(******************************************************************************************************************************************)
(****************************				           Reset Function Part                                                 *****************************)
(******************************************************************************************************************************************)
IF xReset AND NOT(xSetEnd) THEN
	xEnd:=FALSE;
	xSetEnd:=TRUE;
END_IF;
(******************************************************************************************************************************************)
(****************************				              Error Controlling Part                                            *****************************)
(******************************************************************************************************************************************)
IF (xHardwareError OR ((TAxisGrindFeeder.T_CtrleSingle.xErr) AND xStartMainPrc)) AND NOT(xSetEnd) THEN
	IF NOT(TAxisGrindFeeder.T_CtrleSingle.xExecute) THEN
		IF NOT(xInitError) THEN
			iStepError:=100;
			xInitError:=TRUE;
			IF xHardwareError THEN
				iErrorNr:=iTmpErrorNr;
			ELSE
				xHardwareError:=TRUE;	(* Hardware Error *)
			END_IF;
		END_IF;
		CASE iStepError OF
			100:	iStepError:=0;
				xError:=TRUE;
		END_CASE;
		IF xQuitErr THEN
			xSetEnd:=TRUE;
		END_IF;
	END_IF;
END_IF;
(******************************************************************************************************************************************)
(****************************				              Main Controlling Part                                            *****************************)
(******************************************************************************************************************************************)
IF (xStart OR xStartMainCtr) AND NOT(xSetEnd) AND NOT(xHardwareError) THEN
	IF NOT (xInitMainCtr) THEN
		iTmpErrorNr:=0;
		iStepPrc:=100;
		xInitMainCtr:=TRUE;
		xStartMainCtr:=TRUE;
		xStart:=FALSE;
		xEnd:=FALSE;
		xAbord:=FALSE;
		xTmpInit:=FALSE;
	END_IF;
	IF xStop AND NOT(xTmpInit) THEN
		xTmpInit:=TRUE;
		iTmp:=100;
		RETURN;
	END_IF;
	IF xFreeze THEN
		IF xStart AND NOT(xAbord) THEN
			xFreeze:=FALSE;
			xStart:=FALSE;
		END_IF;
		IF xAbord THEN
			xAbord:=FALSE;
			xFreeze:=FALSE;
			xStart:=FALSE;
			xSetEnd:=TRUE;
		END_IF;
		RETURN;
	END_IF;
	IF NOT(xStartMainPrc) AND NOT(xSetEnd) THEN
		xStartMainPrc:=TRUE;
	END_IF;
END_IF;
(******************************************************************************************************************************************)
(****************************				             immediate Stop Part                                              *****************************)
(******************************************************************************************************************************************)
IF xTmpInit AND NOT(xSetEnd) THEN
	IF NOT(xSafetyCircuitOn) THEN
		xTmpInit:=FALSE;
		iTmp:=100;
		xSetEnd:=TRUE;
		RETURN;
	END_IF;
	CASE iTmp OF
		100:	TAxisGrindFeeder.T_CtrleSingle.iFunction:=5;
			TAxisGrindFeeder.T_CtrleSingle.xExecute:=TRUE;
			iTmp:=200;
			RETURN;
		200:	IF NOT(TAxisGrindFeeder.T_CtrleSingle.xExecute) AND TAxisGrindFeeder.T_CtrleSingle.xDone THEN
				iTmp:=300;
			END_IF;
			RETURN;
		300:	xTmpInit:=FALSE;
			iTmp:=100;
			xSetEnd:=TRUE;
			RETURN;
	END_CASE;
END_IF;
(******************************************************************************************************************************************)
(****************************				             Main Procedure Part                                             *****************************)
(******************************************************************************************************************************************)
IF xStartMainPrc AND NOT(xSetEnd) AND NOT(xHardwareError) THEN
	CASE iStepPrc OF
		100:	IF NOT(xInitStep) THEN
				xInitStep:=TRUE;
				IF NOT(TAxisGrindFeeder.T_CtrleSingle.xDone)THEN
					xHardwareError:=TRUE;
					iTmpErrorNr:=1;
					RETURN;
				END_IF;
				IF NOT(TAxisGrindFeeder.T_CtrleSingle.xPower) THEN
					TAxisGrindFeeder.T_CtrleSingle.iFunction:=3;
					TAxisGrindFeeder.T_CtrleSingle.xExecute:=TRUE;
				END_IF;
			END_IF;
			IF NOT(TAxisGrindFeeder.T_CtrleSingle.xExecute) AND TAxisGrindFeeder.T_CtrleSingle.xDone THEN
				xStartMainPrc:=FALSE;
				xInitStep:=FALSE;
				iStepPrc:=200;
			END_IF;
		200:	IF NOT(xInitStep) THEN
				xInitStep:=TRUE;
				IF (iFunctionNr = 4) THEN
					TAxisGrindFeeder.T_CtrleSingle.iFunction:=7;	(* Move Absolut *)
				END_IF;
				IF (iFunctionNr = 5) THEN
					TAxisGrindFeeder.T_CtrleSingle.iFunction:=8;	(* Move Relative *)
				END_IF;
				TAxisGrindFeeder.T_CtrleSingle.xExecute:=TRUE;
			END_IF;
			IF NOT(TAxisGrindFeeder.T_CtrleSingle.xExecute) AND TAxisGrindFeeder.T_CtrleSingle.xDone THEN
				xStartMainPrc:=FALSE;
				xInitStep:=FALSE;
				iStepPrc:=0;
				xSetEnd:=TRUE;
			END_IF;
	END_CASE;
END_IF;
(******************************************************************************************************************************************)
(****************************				           Parallel Procedure Part                                          *****************************)
(******************************************************************************************************************************************)

(******************************************************************************************************************************************)
(****************************				             	Init / Reset Part                                                   *****************************)
(******************************************************************************************************************************************)
IF xSetEnd THEN
	xEnd:=TRUE;
	xInitStep:=FALSE;
	xSetEnd:=FALSE;
	xStop:=FALSE;
	xStartMainPrc:=FALSE;
	xInitMainCtr:=FALSE;
	xStartMainCtr:=FALSE;
	xStart:=FALSE;
	xHardwareError:=FALSE;
	xQuitErr:=FALSE;
	xError:=FALSE;
	iErrorNr:=0;
	xInitError:=FALSE;
	xFreeze:=FALSE;
	xAbord:=FALSE;
	xReset:=FALSE;
END_IF;
END_FUNCTION_BLOCK

(* POU PRG_STATION_LAYER3/FB_STATIONEN/FB_FUNCTION/FB_FctSetAxisPosition, ST *)
FUNCTION_BLOCK FB_FctSetAxisPosition
VAR_INPUT
	xMicroRodActive: BOOL;		(* choice of the machine MicroWire or MicroRod *)
	xBeckhoffDriveActive: BOOL;	(* choice of the axis Beckhoff or EcoStep *)
	xSafetyCircuitOn:BOOL;			(* state of the safety circuit-->TRUE=Machine current ON, FALSE=Machine current OFF *)
	iFunctionNr:INT;				(* state of the called function number-->	6=set position of the ToolLeft axis
																	7=set position of the ToolCenter axis
																	8=set position of the ToolRight axis
																	9=set position of the ToolFeeder axis
																	10=set position of the GrindFeeder axis *)
END_VAR
VAR_IN_OUT
	xStart : BOOL;					(* start the function *)
	xReset : BOOL;				(* reset the function *)
	xStop : BOOL;					(* stop the active function *)
	xQuitErr : BOOL;				(* quit the error caused of the active function *)
	xAbord : BOOL;				(* abord the active function *)
	TAxisToolLeft:ST_AXIS;		(* data structure for the ToolLeft axis *)
	TAxisToolCenter:ST_AXIS;		(* data structure for the ToolCenter axis *)
	TAxisToolRight:ST_AXIS;		(* data structure for the ToolRight axis *)
	TAxisToolFeeder:ST_AXIS;		(* data structure for the ToolFeeder axis *)
	TAxisGrindFeeder:ST_AXIS;	(* data structure for the GrindFeeder axis *)
END_VAR
VAR_OUTPUT
	xEnd : BOOL;					(* state of the function if a active function is ended *)
	xError : BOOL;					(* state of the function if a active function caused an error *)
	iErrorNr : INT;					(* state of the function if a active function caused an error, in this case give the error number *)
END_VAR
VAR
	xHardwareError: BOOL := FALSE;
	xInitError: BOOL := FALSE;
	iStepError: INT := 0;
	xStartMainCtr: BOOL := FALSE;
	xStartMainPrc: BOOL := FALSE;
	xInitMainCtr: BOOL := FALSE;
	iStepPrc: INT := 0;
	xSetEnd: BOOL := FALSE;
	xInitStep: BOOL := FALSE;
	xFreeze: BOOL := FALSE;
	iTmpErrorNr:INT:=0;
	xTmpInit:BOOL;
	iTmp:INT;
	ptrTAxis: POINTER TO ST_AXIS;
	xReadFirstTime: BOOL;
END_VAR
(****************************************************************************************************************************************************)
(***********       This Functionblock set a position for the ToolLeft,ToolCenter,ToolRight,ToolFeeder or GrindFeeder       ************)
(****************************************************************************************************************************************************)

IF NOT(xReadFirstTime) THEN
	xReadFirstTime:=TRUE;
	ptrTAxis:=ADR(TAxisToolLeft);
END_IF;
(******************************************************************************************************************************************)
(****************************				           Reset Function Part                                                 *****************************)
(******************************************************************************************************************************************)
IF xReset AND NOT(xSetEnd) THEN
	ptrTAxis:=ADR(TAxisToolLeft);
	xEnd:=FALSE;
	xSetEnd:=TRUE;
END_IF;
(******************************************************************************************************************************************)
(****************************				              Error Controlling Part                                            *****************************)
(******************************************************************************************************************************************)
IF (xHardwareError OR ((ptrTAxis^.T_CtrleSingle.xErr) AND xStartMainPrc)) AND NOT(xSetEnd) THEN
	IF NOT(ptrTAxis^.T_CtrleSingle.xExecute) THEN
		IF NOT(xInitError) THEN
			iStepError:=100;
			xInitError:=TRUE;
			IF xHardwareError THEN
				iErrorNr:=iTmpErrorNr;
			ELSE
				xHardwareError:=TRUE;	(* Hardware Error *)
			END_IF;
		END_IF;
		CASE iStepError OF
			100:	iStepError:=0;
				xError:=TRUE;
		END_CASE;
		IF xQuitErr THEN
			xSetEnd:=TRUE;
		END_IF;
	END_IF;
END_IF;
(******************************************************************************************************************************************)
(****************************				              Main Controlling Part                                            *****************************)
(******************************************************************************************************************************************)
IF (xStart OR xStartMainCtr) AND NOT(xSetEnd) AND NOT(xHardwareError) THEN
	IF NOT (xInitMainCtr) THEN
		IF (iFunctionNr = 6) THEN
			ptrTAxis:=ADR(TAxisToolLeft);
		ELSIF (iFunctionNr = 7) THEN
			ptrTAxis:=ADR(TAxisToolCenter);
		ELSIF (iFunctionNr = 8) THEN
			ptrTAxis:=ADR(TAxisToolRight);
		ELSIF (iFunctionNr = 9) THEN
			ptrTAxis:=ADR(TAxisToolFeeder);
		ELSIF (iFunctionNr = 10) THEN
			ptrTAxis:=ADR(TAxisGrindFeeder);
		ELSE
			ptrTAxis:=ADR(TAxisToolLeft);
		END_IF;
		iTmpErrorNr:=0;
		iStepPrc:=100;
		xInitMainCtr:=TRUE;
		xStartMainCtr:=TRUE;
		xStart:=FALSE;
		xEnd:=FALSE;
		xAbord:=FALSE;
		xTmpInit:=FALSE;
	END_IF;
	IF xStop AND NOT(xTmpInit) THEN
		xTmpInit:=TRUE;
		iTmp:=100;
		RETURN;
	END_IF;
	IF xFreeze THEN
		IF xStart AND NOT(xAbord) THEN
			xFreeze:=FALSE;
			xStart:=FALSE;
		END_IF;
		IF xAbord THEN
			xAbord:=FALSE;
			xFreeze:=FALSE;
			xStart:=FALSE;
			xSetEnd:=TRUE;
		END_IF;
		RETURN;
	END_IF;
	IF NOT(xStartMainPrc) AND NOT(xSetEnd) THEN
		xStartMainPrc:=TRUE;
	END_IF;
END_IF;
(******************************************************************************************************************************************)
(****************************				             immediate Stop Part                                              *****************************)
(******************************************************************************************************************************************)
IF xTmpInit AND NOT(xSetEnd) THEN
	IF NOT(xSafetyCircuitOn) THEN
		xTmpInit:=FALSE;
		iTmp:=100;
		xSetEnd:=TRUE;
		RETURN;
	END_IF;
	CASE iTmp OF
		100:	IF NOT(ptrTAxis^.T_CtrleSingle.xDone) THEN
				ptrTAxis^.T_CtrleSingle.xReset:=TRUE;
				iTmp:=200;
			END_IF;
			RETURN;
		200:	IF NOT(ptrTAxis^.T_CtrleSingle.xReset) AND ptrTAxis^.T_CtrleSingle.xDone THEN
				iTmp:=300;
			END_IF;
			RETURN;
		300:	xTmpInit:=FALSE;
			iTmp:=100;
			xSetEnd:=TRUE;
			RETURN;
	END_CASE;
END_IF;
(******************************************************************************************************************************************)
(****************************				             Main Procedure Part                                             *****************************)
(******************************************************************************************************************************************)
IF xStartMainPrc AND NOT(xSetEnd) AND NOT(xHardwareError) THEN
	CASE iStepPrc OF
		100:	IF NOT(xInitStep) THEN
				xInitStep:=TRUE;
				IF NOT(ptrTAxis^.T_CtrleSingle.xDone)THEN
					xHardwareError:=TRUE;
					iTmpErrorNr:=1;
					RETURN;
				END_IF;
				ptrTAxis^.T_CtrleSingle.iFunction:=11;
				ptrTAxis^.T_CtrleSingle.xExecute:=TRUE;
			END_IF;
			IF NOT(ptrTAxis^.T_CtrleSingle.xExecute) AND ptrTAxis^.T_CtrleSingle.xDone THEN
				xStartMainPrc:=FALSE;
				xInitStep:=FALSE;
				iStepPrc:=0;
				xSetEnd:=TRUE;
			END_IF;
	END_CASE;
END_IF;
(******************************************************************************************************************************************)
(****************************				           Parallel Procedure Part                                          *****************************)
(******************************************************************************************************************************************)

(******************************************************************************************************************************************)
(****************************				             	Init / Reset Part                                                   *****************************)
(******************************************************************************************************************************************)
IF xSetEnd THEN
	xEnd:=TRUE;
	xInitStep:=FALSE;
	xSetEnd:=FALSE;
	xStop:=FALSE;
	xStartMainPrc:=FALSE;
	xInitMainCtr:=FALSE;
	xStartMainCtr:=FALSE;
	xStart:=FALSE;
	xHardwareError:=FALSE;
	xQuitErr:=FALSE;
	xError:=FALSE;
	iErrorNr:=0;
	xInitError:=FALSE;
	xFreeze:=FALSE;
	xAbord:=FALSE;
	xReset:=FALSE;
END_IF;
END_FUNCTION_BLOCK

(* POU PRG_STATION_LAYER3/FB_STATIONEN/FB_FUNCTION/FB_FctToolWorkingGeometry, ST *)
FUNCTION_BLOCK FB_FctToolWorkingGeometry
VAR_INPUT
	xMicroRodActive: BOOL;		(* choice of the machine MicroWire or MicroRod *)
	xBeckhoffDriveActive: BOOL;	(* choice of the axis Beckhoff or EcoStep *)
	xSafetyCircuitOn:BOOL;			(* state of the safety circuit-->TRUE=Machine current ON, FALSE=Machine current OFF *)
	T_ProcessImageData:ST_RETAIN_DATA_PROCESSIMAGE;	(* Novram data structure for the process parameter *)
	T_Standard:ST_RETAIN_DATA;							(* Novram data structure for the standard process parameter *)
END_VAR
VAR_IN_OUT
	xStart : BOOL;					(* start the function *)
	xReset : BOOL;				(* reset the function *)
	xStop : BOOL;					(* stop the active function *)
	xQuitErr : BOOL;				(* quit the error caused of the active function *)
	xAbord : BOOL;				(* abord the active function *)
	TAxisToolLeft:ST_AXIS;		(* data structure for the ToolLeft axis *)
	TAxisToolCenter:ST_AXIS;		(* data structure for the ToolCenter axis *)
	TAxisToolRight:ST_AXIS;		(* data structure for the ToolRight axis *)
	TAxisToolFeeder:ST_AXIS;		(* data structure for the ToolFeeder axis *)
	TAxisGrindFeeder:ST_AXIS;	(* data structure for the GrindFeeder axis *)
	T_WorkTool:ST_WORKTOOL;	(* Tool parameter *)
END_VAR
VAR_OUTPUT
	xEnd : BOOL;					(* state of the function if a active function is ended *)
	xError : BOOL;					(* state of the function if a active function caused an error *)
	iErrorNr : INT;					(* state of the function if a active function caused an error, in this case give the error number *)
	bActivePartNumber:BYTE;		(* gives the active number of the worked section of the geometry *)
	lrProcessToolFeederActualPosition:LREAL;	(* gives the calculated position of the ToolFeeder *)
	lrProcessToolFeederSpeed:LREAL;			(* gives the calculated speed of the ToolFeeder *)
	iCountDownPlungeCycle:INT;
END_VAR
VAR
	xHardwareError: BOOL := FALSE;
	xInitError: BOOL := FALSE;
	iStepError: INT := 0;
	xStartMainCtr: BOOL := FALSE;
	xStartMainPrc: BOOL := FALSE;
	xInitMainCtr: BOOL := FALSE;
	iStepPrc: INT := 0;
	xSetEnd: BOOL := FALSE;
	xInitStep: BOOL := FALSE;
	xFreeze: BOOL := FALSE;
	iTmpErrorNr:INT:=0;
	xTmpInit:BOOL;
	iTmp:INT;
	xTmp: BOOL;
	xReadFirstTime: BOOL;
	xTmp1: BOOL;
	rToolRotationSpeed: REAL;
	FBToolCalcul:FB_TOOL_CALCUL_NEW;

	rToolFeedLength: REAL;
	rToolDiameter: REAL;
	rGrindFeedPlunge: REAL;
	ii: INT;
	iStartSection: INT;
	iEndSection: INT;
	rSpeedGrindFeed: REAL;
	rSpeedToolFeed: REAL;
	rTimeGrindPlunge: REAL;
	FBCalcGearFactor: FB_CALC_GEARFACTOR;
	lrToolFeederActualPosition: LREAL;
	iTmpStartSection: INT;
	FBCalcPlungeGrinding: FB_CALC_PLUNGE_GRINDING;
	xResetFB: BOOL;
	xGrindFeedMaster: BOOL;
	xCheckToolFeedPosition: BOOL;
	lrToolFeederPosition: LREAL;
	lrToolRightPosition: LREAL;
	lrSaveToolFeederPosition: LREAL;
	lrSaveToolRightPosition: LREAL;
	rPlungeCycleGrindFeedGeometry: REAL;
	lrGearFactor: LREAL;
	xPositionReached: BOOL;
	lrToolFeedCalcLengthPosition: REAL;
	lrCalcToolLengthInc: LREAL;
	lrCalcToolLength: LREAL;
	xReadyToolFeedStop: BOOL;
	xReadyGrindFeedStop: BOOL;
END_VAR
(****************************************************************************************************************************************************)
(***********                                This Functionblock define the function for work a geometry on the tool                                          ************)
(****************************************************************************************************************************************************)

IF NOT(xReadFirstTime) THEN
	xReadFirstTime:=TRUE;
END_IF;
(******************************************************************************************************************************************)
(****************************				           Reset Function Part                                                 *****************************)
(******************************************************************************************************************************************)
IF xReset AND NOT(xSetEnd) THEN
	xEnd:=FALSE;
	xSetEnd:=TRUE;
END_IF;
(******************************************************************************************************************************************)
(****************************				              Error Controlling Part                                            *****************************)
(******************************************************************************************************************************************)
xTmp:=	TAxisToolLeft.T_CtrleSingle.xErr OR
		(TAxisToolCenter.T_CtrleSingle.xErr AND xMicroRodActive) OR
		TAxisToolRight.T_CtrleSingle.xErr OR
		TAxisToolFeeder.T_CtrleSingle.xErr OR
		TAxisGrindFeeder.T_CtrleSingle.xErr;
xTmp1:=	NOT(TAxisToolLeft.T_CtrleSingle.xExecute) AND
		((NOT(TAxisToolCenter.T_CtrleSingle.xExecute) AND xMicroRodActive) OR NOT(xMicroRodActive)) AND
		 NOT(TAxisToolRight.T_CtrleSingle.xExecute) AND
		((NOT(TAxisToolFeeder.T_CtrleSingle.xExecute) AND NOT(xMicroRodActive)) OR xMicroRodActive) AND
		NOT(TAxisGrindFeeder.T_CtrleSingle.xExecute);
IF (xHardwareError OR (xTmp AND xStartMainPrc)) AND NOT(xSetEnd) THEN
	IF xTmp1 THEN
		IF NOT(xInitError) THEN
			iStepError:=100;
			xInitError:=TRUE;
			IF xHardwareError THEN
				iErrorNr:=iTmpErrorNr;
			ELSE
				xHardwareError:=TRUE;	(* Hardware Error *)
			END_IF;
		END_IF;
		CASE iStepError OF
			100:	iStepError:=0;
				xError:=TRUE;
		END_CASE;
		IF xQuitErr THEN
			xSetEnd:=TRUE;
		END_IF;
	END_IF;
END_IF;
(******************************************************************************************************************************************)
(****************************				              Main Controlling Part                                            *****************************)
(******************************************************************************************************************************************)
IF (xStart OR xStartMainCtr) AND NOT(xSetEnd) AND NOT(xHardwareError) THEN
	IF NOT (xInitMainCtr) THEN
		iTmpErrorNr:=0;
		iStepPrc:=100;
		xInitMainCtr:=TRUE;
		xStartMainCtr:=TRUE;
		xStart:=FALSE;
		xEnd:=FALSE;
		xAbord:=FALSE;
		xTmpInit:=FALSE;
		xCheckToolFeedPosition:=FALSE;
		bActivePartNumber:=0;
		lrCalcToolLengthInc:=lrCalcToolLength:=0.0;
		rSpeedToolFeed:=0.0;
		iCountDownPlungeCycle:=1;
	END_IF;
	IF xStop AND NOT(xTmpInit) THEN
		xTmpInit:=TRUE;
		iTmp:=100;
		RETURN;
	END_IF;
	IF xFreeze THEN
		IF xStart AND NOT(xAbord) THEN
			xFreeze:=FALSE;
			xStart:=FALSE;
		END_IF;
		IF xAbord THEN
			xAbord:=FALSE;
			xFreeze:=FALSE;
			xStart:=FALSE;
			xSetEnd:=TRUE;
		END_IF;
		RETURN;
	END_IF;
	IF NOT(xStartMainPrc) AND NOT(xSetEnd) THEN
		xStartMainPrc:=TRUE;
	END_IF;
END_IF;
(******************************************************************************************************************************************)
(****************************		               Controlling of the ToolFeeder Position                            *****************************)
(******************************************************************************************************************************************)
IF xCheckToolFeedPosition THEN
	IF xMicroRodActive THEN
		lrToolFeederPosition:=TAxisToolFeeder.T_LiveValue.lrActualPositionNotModulo - lrSaveToolFeederPosition;
		lrToolFeederActualPosition:=(lrToolFeederPosition / TAxisToolFeeder.T_CtrleSingle.lrScaleFactor);
		lrCalcToolLength:=lrToolFeederActualPosition;
	END_IF;
	IF NOT(xMicroRodActive) AND (TAxisToolRight.T_CtrleSingle.lrGearRatio <> 0.0) THEN
		lrToolFeedCalcLengthPosition:=((((T_WorkTool.rToolLength * 10.0) / ABS(T_WorkTool.rPitch)) * 24000.0) / TAxisToolRight.T_CtrleSingle.lrScaleFactor);
		lrToolFeederPosition:=lrToolFeederPosition + ABS(ABS(TAxisToolRight.T_LiveValue.lrActualPosition) - (lrSaveToolFeederPosition / TAxisToolRight.T_CtrleSingle.lrScaleFactor));
		lrSaveToolFeederPosition:=ABS(TAxisToolRight.T_LiveValue.lrActualPositionNotModulo);
		lrToolFeederActualPosition:=((T_WorkTool.rToolLength * 10.0) / lrToolFeedCalcLengthPosition) * lrToolFeederPosition;
		lrCalcToolLength:=lrCalcToolLengthInc + lrToolFeederActualPosition;
	END_IF;
ELSE
	IF NOT(xMicroRodActive) AND (TAxisToolRight.T_CtrleSingle.lrGearRatio <> 0.0) THEN
		lrSaveToolFeederPosition:=ABS(TAxisToolRight.T_LiveValue.lrActualPositionNotModulo);
		lrSaveToolRightPosition:=TAxisToolRight.T_LiveValue.lrActualPositionNotModulo * TAxisToolRight.T_CtrleSingle.lrGearRatio;
		lrCalcToolLengthInc:=lrCalcToolLength;
	END_IF;
	IF xMicroRodActive THEN
		lrSaveToolFeederPosition:=TAxisToolFeeder.T_LiveValue.lrActualPositionNotModulo;
	END_IF;
	lrToolFeederActualPosition:=lrToolFeederPosition:=0.0;
END_IF;
lrProcessToolFeederActualPosition:=lrCalcToolLength;
lrProcessToolFeederSpeed:=rSpeedToolFeed;
(******************************************************************************************************************************************)
(****************************				             immediate Stop Part                                              *****************************)
(******************************************************************************************************************************************)
IF xTmpInit AND NOT(xSetEnd) THEN
	IF NOT(xSafetyCircuitOn) THEN
		xTmpInit:=FALSE;
		iTmp:=100;
		xSetEnd:=TRUE;
		RETURN;
	END_IF;
	CASE iTmp OF
		100:	xReadyToolFeedStop:=xReadyGrindFeedStop:=FALSE;
			TAxisGrindFeeder.T_CtrleSingle.lrAcceleration:=T_Standard.T_TeachINToolFeeder.rAcceleration;
			TAxisGrindFeeder.T_CtrleSingle.lrDecceleration:=T_Standard.T_TeachINToolFeeder.rDeceleration;
			TAxisGrindFeeder.T_CtrleSingle.iFunction:=5;	(* Stop Movement *)
			TAxisGrindFeeder.T_CtrleSingle.xExecute:=TRUE;
			iTmp:=200;
			RETURN;
		200:	IF NOT(TAxisGrindFeeder.T_CtrleSingle.xExecute) AND TAxisGrindFeeder.T_CtrleSingle.xDone THEN
				TAxisGrindFeeder.T_CtrleSingle.lrAcceleration:=T_Standard.T_TeachINGrindFeeder.rAcceleration;
				TAxisGrindFeeder.T_CtrleSingle.lrDecceleration:=T_Standard.T_TeachINGrindFeeder.rDeceleration;
				TAxisGrindFeeder.T_CtrleSingle.lrPosition:=	T_ProcessImageData.T_ProcessPara.rToolDiameterProcess +
														T_ProcessImageData.T_ProcessPara.rSecurityPosGrindFeedProcess;
				TAxisGrindFeeder.T_CtrleSingle.lrVelocity:=T_ProcessImageData.T_ProcessPara.rSpeedBackwardGrindFeed;
				TAxisGrindFeeder.T_CtrleSingle.iFunction:=7;	(* Move Absolut *)
				TAxisGrindFeeder.T_CtrleSingle.xExecute:=TRUE;
				iTmp:=300;
			END_IF;
			RETURN;
		300:	IF NOT(TAxisGrindFeeder.T_CtrleSingle.xExecute) AND TAxisGrindFeeder.T_CtrleSingle.xDone AND NOT(xReadyGrindFeedStop) THEN
				xReadyGrindFeedStop:=TRUE;
			END_IF;
			IF (TAxisGrindFeeder.T_LiveValue.lrActualPosition >= (T_ProcessImageData.T_ProcessPara.rToolDiameterProcess + T_ProcessImageData.T_ProcessPara.rOffsetBeforeToolDiaGrindFeedProcess)) AND NOT(xReadyToolFeedStop) THEN
				xReadyToolFeedStop:=TRUE;
				xCheckToolFeedPosition:=FALSE;
				IF xMicroRodActive THEN
					IF NOT(TAxisToolFeeder.T_CtrleSingle.xNotMoving) THEN
						TAxisToolFeeder.T_CtrleSingle.lrAcceleration:=T_Standard.T_TeachINToolFeeder.rAcceleration;
						TAxisToolFeeder.T_CtrleSingle.lrDecceleration:=T_Standard.T_TeachINToolFeeder.rDeceleration;
						TAxisToolFeeder.T_CtrleSingle.iFunction:=5;	(* Stop Movement *)
						TAxisToolFeeder.T_CtrleSingle.xExecute:=TRUE;
					END_IF;
				END_IF;
				IF NOT(xMicroRodActive) THEN
					FBCalcGearFactor(	rSpeed:= 0.0,
										rToolRotationSpeed:= rToolRotationSpeed,
										T_WorkTool:=T_WorkTool );
					TAxisToolFeeder.T_CtrleSingle.lrGearFactor:=INT_TO_LREAL(FBCalcGearFactor.T_WorkTool.iToolFeederGearFactor) * -1.0;
					TAxisToolFeeder.T_CtrleSingle.lrGearDivider:=INT_TO_LREAL(FBCalcGearFactor.T_WorkTool.iToolFeederGearDivider);
					(* Set Gear Value with PDO Object *)
					TAxisToolFeeder.T_RxPdoParameter.iGearFactor:=LREAL_TO_INT(TAxisToolFeeder.T_CtrleSingle.lrGearFactor);
					TAxisToolFeeder.T_RxPdoParameter.uiGearDivider:=LREAL_TO_UINT(TAxisToolFeeder.T_CtrleSingle.lrGearDivider);
				END_IF;
				lrProcessToolFeederSpeed:=0.0;
			END_IF;
			IF xReadyToolFeedStop AND xReadyGrindFeedStop THEN
				iTmp:=400;
			END_IF;
			RETURN;
		400:	IF NOT(TAxisToolFeeder.T_CtrleSingle.xExecute) AND TAxisToolFeeder.T_CtrleSingle.xDone THEN
				iTmp:=500;
			END_IF;
			RETURN;
		500:	xTmpInit:=FALSE;
			iTmp:=100;
			xSetEnd:=TRUE;
			RETURN;
	END_CASE;
END_IF;
(******************************************************************************************************************************************)
(****************************				             Main Procedure Part                                             *****************************)
(******************************************************************************************************************************************)
IF xStartMainPrc AND NOT(xSetEnd) AND NOT(xHardwareError) THEN
	CASE iStepPrc OF
		(* Initial Procedure *)
		100:	rToolFeedLength:=0.0;
			rToolDiameter:=T_ProcessImageData.T_ProcessPara.rToolDiameterProcess;
			rGrindFeedPlunge:=0.0;
			rSpeedGrindFeed:=0.0;
			rSpeedToolFeed:=0.0;
			iStartSection:=1;
			(* Check Start and End Section of the ToolGeometry *)
			FOR ii:=1 TO 6 DO
				IF T_ProcessImageData.T_GeometryPara.axActiveSection[ii] THEN
					IF (iStartSection = 0) THEN
						iStartSection:=ii;
					END_IF;
					iEndSection:=ii;
				END_IF;
			END_FOR;
			xResetFB:=TRUE;
			FBCalcPlungeGrinding(	rToolDiameter:= T_ProcessImageData.T_ProcessPara.rToolDiameterProcess,
									rToolDiameterWithOffset:=T_ProcessImageData.T_ProcessPara.rToolDiameterProcess + T_ProcessImageData.T_ProcessPara.rOffsetBeforeToolDiaGrindFeedProcess,
									xReset:= xResetFB);
			IF xMicroRodActive THEN
				rPlungeCycleGrindFeedGeometry:=T_ProcessImageData.T_AutoGeometryPara.rPlungeCycleGrindFeedGeometry;
			END_IF;
			IF NOT(xMicroRodActive) THEN
			(* MicroWire is not aloved to work in more cycle *)
				rPlungeCycleGrindFeedGeometry:=T_ProcessImageData.T_ProcessPara.rToolDiameterProcess;
			END_IF;
			xStartMainPrc:=FALSE;
			xInitStep:=FALSE;
			(* Start with AutoGeometry working *)
			iStepPrc:=200;
		(* Calculation of Grind plunge of all section, include Plunge procedure and Displace procedure *)
		200:	IF NOT(xInitStep) THEN
				xInitStep:=TRUE;
				FBCalcPlungeGrinding(	T_Geometry:= T_ProcessImageData.T_GeometryPara,
										T_AutoGeometryPara:= T_ProcessImageData.T_AutoGeometryPara,
										rToolDiameter:= T_ProcessImageData.T_ProcessPara.rToolDiameterProcess,
										rToolDiameterWithOffset:=T_ProcessImageData.T_ProcessPara.rToolDiameterProcess + T_ProcessImageData.T_ProcessPara.rOffsetBeforeToolDiaGrindFeedProcess,
										rPlungeCycleGrindFeedGeometry:=rPlungeCycleGrindFeedGeometry,
										iStartSection:= iStartSection,
										iEndSection:= iEndSection,
										xReset:= xResetFB);
			END_IF;
			IF xInitStep THEN
				bActivePartNumber:=INT_TO_BYTE(FBCalcPlungeGrinding.iStepSectionWork);
				xStartMainPrc:=FALSE;
				xInitStep:=FALSE;
				IF FBCalcPlungeGrinding.xEndWorking THEN
					iStepPrc:=400;
				ELSE
					iStepPrc:=300;
				END_IF;
			END_IF;
		300:	IF NOT(xInitStep) THEN
				xInitStep:=TRUE;
				xGrindFeedMaster:=FALSE;
	(********************************                              Plunge Procedure                         *******************************)
				IF (FBCalcPlungeGrinding.iStepSectionWork = 0) THEN
					rToolFeedLength:=0.0;
					rSpeedToolFeed:=0.0;
					IF T_ProcessImageData.T_AutoGeometryPara.xPlungeActivationGeometry THEN
						rToolFeedLength:=T_ProcessImageData.T_AutoGeometryPara.rPlungeLengthToolFeedGeometry;
						T_WorkTool.rToolLength:=rToolFeedLength/10.0;
					ELSE
						T_WorkTool.rToolLength:=0.0;
					END_IF;
					IF T_ProcessImageData.T_AutoGeometryPara.xPlungeActivationGeometry THEN
						T_WorkTool.rToolRotationSpeed:=T_ProcessImageData.T_AutoGeometryPara.rSpeedToolRotationGeometry;
						T_WorkTool.rPitch:=T_ProcessImageData.T_GeometryPara.arSectionPitch[iStartSection] * -1.0;
						T_WorkTool.rGrindFeederPlunge:=	FBCalcPlungeGrinding.rGrindingRelativePosition;
						FBToolCalcul(	xMicroRodActive:=xMicroRodActive,
										xBeckhoffDriveActive:=FALSE,
										T_WorkTool:= T_WorkTool,
										rToolFeedAcclDecl:= T_Standard.T_TeachINToolFeeder.rAcceleration);
						rGrindFeedPlunge:=T_WorkTool.rGrindFeederPlunge * -1.0;
						rSpeedGrindFeed:=T_WorkTool.rGrindFeederSpeedUnit;
						rSpeedToolFeed:=T_WorkTool.rToolFeederSpeedUnit * -1.0;
					ELSE
						rSpeedGrindFeed:=T_ProcessImageData.T_AutoGeometryPara.rPlungeSpeedGrindFeedGeometry;
						rGrindFeedPlunge:=FBCalcPlungeGrinding.rGrindingRelativePosition * -1.0;
						IF (rToolFeedLength <> 0) THEN
							rTimeGrindPlunge:=ABS(rGrindFeedPlunge) / rSpeedGrindFeed;		(* calc Time in seocnds *)
							rSpeedToolFeed:=rToolFeedLength / rTimeGrindPlunge;	(* calc Speed ToolFeed in mm/s *)
						END_IF;
						T_WorkTool.rPitch:=T_ProcessImageData.T_GeometryPara.arSectionPitch[iStartSection] * -1.0;
					END_IF;
					rToolRotationSpeed:=T_ProcessImageData.T_AutoGeometryPara.rSpeedToolRotationGeometry;
				END_IF;
	(********************************                              Geometry Procedure                         *******************************)
				IF (FBCalcPlungeGrinding.iStepSectionWork > 0) AND (FBCalcPlungeGrinding.iStepSectionWork < 7) THEN
					(* Check first active section *)
					iTmpStartSection:=iStartSection + (FBCalcPlungeGrinding.iStepSectionWork - 1);
					T_WorkTool.rToolRotationSpeed:=T_ProcessImageData.T_AutoGeometryPara.rSpeedToolRotationGeometry;
					T_WorkTool.rPitch:=T_ProcessImageData.T_GeometryPara.arSectionPitch[iTmpStartSection] * -1.0;
					T_WorkTool.rToolLength:=T_ProcessImageData.T_GeometryPara.arSectionLength[iTmpStartSection];
					rGrindFeedPlunge:=FBCalcPlungeGrinding.rGrindingRelativePosition * -1.0;
					T_WorkTool.rGrindFeederPlunge:=rGrindFeedPlunge;
					FBToolCalcul(	xMicroRodActive:=xMicroRodActive,
									xBeckhoffDriveActive:=FALSE,
									T_WorkTool:= T_WorkTool,
									rToolFeedAcclDecl:= 0);
					rSpeedGrindFeed:=T_WorkTool.rGrindFeederSpeedUnit;
					rToolFeedLength:=T_WorkTool.rToolLength;
					rSpeedToolFeed:=T_WorkTool.rToolFeederSpeedUnit;
					rToolRotationSpeed:=T_WorkTool.rToolRotationSpeed;
				END_IF;
	(********************************                              Displace Procedure                         *******************************)
				IF (FBCalcPlungeGrinding.iStepSectionWork = 7) THEN
					rToolFeedLength:=0.0;
					rSpeedToolFeed:=0.0;
					IF T_ProcessImageData.T_AutoGeometryPara.xDisplaceActivationGeometry THEN
						rToolFeedLength:=T_ProcessImageData.T_AutoGeometryPara.rDisplaceLengthToolFeedGeometry;
						T_WorkTool.rToolLength:=rToolFeedLength/10.0;
					ELSE
						T_WorkTool.rToolLength:=0.0;
					END_IF;
					IF T_ProcessImageData.T_AutoGeometryPara.xDisplaceActivationGeometry THEN
						T_WorkTool.rToolRotationSpeed:=T_ProcessImageData.T_AutoGeometryPara.rSpeedToolRotationGeometry;
						T_WorkTool.rPitch:=T_ProcessImageData.T_GeometryPara.arSectionPitch[iEndSection] * -1.0;
						T_WorkTool.rGrindFeederPlunge:=	FBCalcPlungeGrinding.rGrindingRelativePosition * -1.0;
						FBToolCalcul(	xMicroRodActive:=xMicroRodActive,
										xBeckhoffDriveActive:=FALSE,
										T_WorkTool:= T_WorkTool,
										rToolFeedAcclDecl:= 0);
						rGrindFeedPlunge:=T_WorkTool.rGrindFeederPlunge;
						rSpeedGrindFeed:=T_WorkTool.rGrindFeederSpeedUnit;
						rSpeedToolFeed:=T_WorkTool.rToolFeederSpeedUnit * -1.0;
					ELSE
						rSpeedGrindFeed:=T_ProcessImageData.T_AutoGeometryPara.rDisplaceSpeedGrindFeedGeometry;
						rGrindFeedPlunge:=FBCalcPlungeGrinding.rGrindingRelativePosition * -1.0;
						IF (rToolFeedLength <> 0) THEN
							rTimeGrindPlunge:=ABS(rGrindFeedPlunge) / rSpeedGrindFeed;		(* calc Time in seocnds *)
							rSpeedToolFeed:=(rToolFeedLength * 10.0) / rTimeGrindPlunge;	(* calc Speed ToolFeed in mm/s *)
						END_IF;
						T_WorkTool.rPitch:=T_ProcessImageData.T_GeometryPara.arSectionPitch[iEndSection] * -1.0;
					END_IF;
					rToolRotationSpeed:=T_ProcessImageData.T_AutoGeometryPara.rSpeedToolRotationGeometry;
				END_IF;
	(********************************                              Drive Procedure                             *******************************)
				IF xMicroRodActive THEN
					IF (*TAxisToolFeeder.T_CtrleSingle.xNotMoving AND*) (rToolFeedLength <> 0) THEN
						TAxisToolFeeder.T_CtrleSingle.lrAcceleration:=T_Standard.T_TeachINToolFeeder.rAcceleration;
						TAxisToolFeeder.T_CtrleSingle.lrDecceleration:=T_Standard.T_TeachINToolFeeder.rDeceleration;
						IF (FBCalcPlungeGrinding.iStepSectionWork > 0) AND (FBCalcPlungeGrinding.iStepSectionWork < 5) THEN
							TAxisToolFeeder.T_CtrleSingle.lrVelocity:=rSpeedToolFeed * -1.0;
						ELSE
							TAxisToolFeeder.T_CtrleSingle.lrVelocity:=rSpeedToolFeed;
						END_IF;
						TAxisToolFeeder.T_CtrleSingle.iFunction:=6;	(* Move continue velocity *)
						TAxisToolFeeder.T_CtrleSingle.xExecute:=TRUE;
					END_IF;
					IF NOT(TAxisToolFeeder.T_CtrleSingle.xNotMoving) AND (rToolFeedLength = 0) THEN
						TAxisToolFeeder.T_CtrleSingle.lrAcceleration:=T_Standard.T_TeachINToolFeeder.rAcceleration;
						TAxisToolFeeder.T_CtrleSingle.lrDecceleration:=T_Standard.T_TeachINToolFeeder.rDeceleration;
						TAxisToolFeeder.T_CtrleSingle.iFunction:=5;	(* Stop Movement *)
						TAxisToolFeeder.T_CtrleSingle.xExecute:=TRUE;
					END_IF;
				END_IF;
				IF NOT(xMicroRodActive) THEN
					IF (FBCalcPlungeGrinding.iStepSectionWork < 1) OR (FBCalcPlungeGrinding.iStepSectionWork > 6) THEN
						FBCalcGearFactor(	rSpeed:= rSpeedToolFeed * -1.0,
											rToolRotationSpeed:= rToolRotationSpeed,
											T_WorkTool:=T_WorkTool );
						TAxisToolFeeder.T_CtrleSingle.lrGearFactor:=INT_TO_LREAL(FBCalcGearFactor.T_WorkTool.iToolFeederGearFactor) * -1.0;
						TAxisToolFeeder.T_CtrleSingle.lrGearDivider:=INT_TO_LREAL(FBCalcGearFactor.T_WorkTool.iToolFeederGearDivider);
					ELSE
						TAxisToolFeeder.T_CtrleSingle.lrGearFactor:=INT_TO_LREAL(T_WorkTool.iToolFeederGearFactor) * -1.0;
						TAxisToolFeeder.T_CtrleSingle.lrGearDivider:=INT_TO_LREAL(T_WorkTool.iToolFeederGearDivider);
					END_IF;
					(* Set Gear Value with PDO Object *)
					TAxisToolFeeder.T_RxPdoParameter.iGearFactor:=LREAL_TO_INT(TAxisToolFeeder.T_CtrleSingle.lrGearFactor);
					TAxisToolFeeder.T_RxPdoParameter.uiGearDivider:=LREAL_TO_UINT(TAxisToolFeeder.T_CtrleSingle.lrGearDivider);
				END_IF;
				(* Start GrindFeeder *)
				IF (rGrindFeedPlunge <> 0) THEN
					xGrindFeedMaster:=TRUE;
					IF (rToolFeedLength <> 0) THEN
						xCheckToolFeedPosition:=TRUE;	(* Start Measure Relative Position of the ToolFeeder *)
					END_IF;
					IF (FBCalcPlungeGrinding.iStepSectionWork > 0) THEN
						TAxisGrindFeeder.T_CtrleSingle.xBlockAcclDeclParameter:=TRUE;	(* do not send again the accl and decl parameter-->better performance *)
					END_IF;
					TAxisGrindFeeder.T_CtrleSingle.lrAcceleration:=T_Standard.T_TeachINGrindFeeder.rAcceleration;
					TAxisGrindFeeder.T_CtrleSingle.lrDecceleration:=T_Standard.T_TeachINGrindFeeder.rDeceleration;
					TAxisGrindFeeder.T_CtrleSingle.lrDistance:=rGrindFeedPlunge;
					TAxisGrindFeeder.T_CtrleSingle.lrVelocity:=rSpeedGrindFeed;
					TAxisGrindFeeder.T_CtrleSingle.iFunction:=8;	(* Move Relative *)
					TAxisGrindFeeder.T_CtrleSingle.xExecute:=TRUE;
				ELSE
					xGrindFeedMaster:=FALSE;
					xCheckToolFeedPosition:=TRUE;	(* Start Measure Relative Position of the ToolFeeder *)
				END_IF;
			END_IF;
	(********************************                              Wait end active section                             *******************************)
			IF xGrindFeedMaster THEN
			(* This is active by plunge procedure or displace procedure or by work a cone section *)
				IF NOT(TAxisGrindFeeder.T_CtrleSingle.xExecute) AND TAxisGrindFeeder.T_CtrleSingle.xDone THEN
					xCheckToolFeedPosition:=FALSE;
					xStartMainPrc:=FALSE;
					xInitStep:=FALSE;
					IF (FBCalcPlungeGrinding.iStepSectionWork <> 7) THEN
						iStepPrc:=200;
					ELSE
						IF xMicroRodActive THEN
							iStepPrc:=400;
						ELSE
							iStepPrc:=200;
						END_IF;
					END_IF;
				END_IF;
			END_IF;
			IF NOT(xGrindFeedMaster) THEN
			(* This is only active if it is work a cylinder section *)
				IF (lrToolFeederActualPosition > (rToolFeedLength * 10.0)) THEN
					xCheckToolFeedPosition:=FALSE;
					xStartMainPrc:=FALSE;
					xInitStep:=FALSE;
					IF (FBCalcPlungeGrinding.iStepSectionWork <> 7) THEN
						iStepPrc:=200;
					ELSE
						IF xMicroRodActive THEN
							iStepPrc:=400;
						ELSE
							iStepPrc:=200;
						END_IF;
					END_IF;
				END_IF;
			END_IF;
		(* Check if ToolFeeder Moves and stop it if it moves *)
		400:	IF NOT(xInitStep) THEN
				xInitStep:=TRUE;
				IF xMicroRodActive THEN
					IF NOT(TAxisToolFeeder.T_CtrleSingle.xNotMoving) THEN
						TAxisToolFeeder.T_CtrleSingle.lrAcceleration:=T_Standard.T_TeachINToolFeeder.rAcceleration;
						TAxisToolFeeder.T_CtrleSingle.lrDecceleration:=T_Standard.T_TeachINToolFeeder.rDeceleration;
						TAxisToolFeeder.T_CtrleSingle.iFunction:=5;	(* Stop Movement *)
						TAxisToolFeeder.T_CtrleSingle.xExecute:=TRUE;
					END_IF;
				END_IF;
				IF NOT(xMicroRodActive) THEN
					FBCalcGearFactor(	rSpeed:= 0.0,
										rToolRotationSpeed:= rToolRotationSpeed,
										T_WorkTool:=T_WorkTool );
					TAxisToolFeeder.T_CtrleSingle.lrGearFactor:=INT_TO_LREAL(FBCalcGearFactor.T_WorkTool.iToolFeederGearFactor) * -1.0;
					TAxisToolFeeder.T_CtrleSingle.lrGearDivider:=INT_TO_LREAL(FBCalcGearFactor.T_WorkTool.iToolFeederGearDivider);
					(* Set Gear Value with PDO Object *)
					TAxisToolFeeder.T_RxPdoParameter.iGearFactor:=LREAL_TO_INT(TAxisToolFeeder.T_CtrleSingle.lrGearFactor);
					TAxisToolFeeder.T_RxPdoParameter.uiGearDivider:=LREAL_TO_UINT(TAxisToolFeeder.T_CtrleSingle.lrGearDivider);
				END_IF;
			END_IF;
			IF NOT(TAxisToolFeeder.T_CtrleSingle.xExecute) AND TAxisToolFeeder.T_CtrleSingle.xDone THEN
				rSpeedToolFeed:=0.0;
				xStartMainPrc:=FALSE;
				xInitStep:=FALSE;
				iStepPrc:=500;
			END_IF;
		(* GrindFeeder go to Security Position *)
		500:	IF NOT(xInitStep) THEN
				xInitStep:=TRUE;
				TAxisGrindFeeder.T_CtrleSingle.lrAcceleration:=T_Standard.T_TeachINGrindFeeder.rAcceleration;
				TAxisGrindFeeder.T_CtrleSingle.lrDecceleration:=T_Standard.T_TeachINGrindFeeder.rDeceleration;
				TAxisGrindFeeder.T_CtrleSingle.lrPosition:=	T_ProcessImageData.T_ProcessPara.rToolDiameterProcess +
														T_ProcessImageData.T_ProcessPara.rSecurityPosGrindFeedProcess;
				TAxisGrindFeeder.T_CtrleSingle.lrVelocity:=T_ProcessImageData.T_ProcessPara.rSpeedBackwardGrindFeed;
				TAxisGrindFeeder.T_CtrleSingle.iFunction:=7;	(* Move Absolut *)
				TAxisGrindFeeder.T_CtrleSingle.xExecute:=TRUE;
			END_IF;
			IF NOT(TAxisGrindFeeder.T_CtrleSingle.xExecute) AND TAxisGrindFeeder.T_CtrleSingle.xDone THEN
				IF FBCalcPlungeGrinding.xEndWorking THEN
					(* Procedure is finished *)
					xStartMainPrc:=FALSE;
					xInitStep:=FALSE;
					iStepPrc:=900;
				ELSE
					(* Only for MicroRod --> Work next cycle *)
					xStartMainPrc:=FALSE;
					xInitStep:=FALSE;
					iStepPrc:=600;
				END_IF;
			END_IF;
		(* Calculation of Grind plunge of all section, include Plunge procedure and Displace procedure *)
		600:	IF NOT(xInitStep) THEN
				xInitStep:=TRUE;
				FBCalcPlungeGrinding(	T_Geometry:= T_ProcessImageData.T_GeometryPara,
										T_AutoGeometryPara:= T_ProcessImageData.T_AutoGeometryPara,
										rToolDiameter:= T_ProcessImageData.T_ProcessPara.rToolDiameterProcess,
										rToolDiameterWithOffset:=T_ProcessImageData.T_ProcessPara.rToolDiameterProcess + T_ProcessImageData.T_ProcessPara.rOffsetBeforeToolDiaGrindFeedProcess,
										rPlungeCycleGrindFeedGeometry:=rPlungeCycleGrindFeedGeometry,
										iStartSection:= iStartSection,
										iEndSection:= iEndSection,
										xReset:= xResetFB);
			END_IF;
			IF xInitStep THEN
				bActivePartNumber:=INT_TO_BYTE(FBCalcPlungeGrinding.iStepSectionWork);
				xStartMainPrc:=FALSE;
				xInitStep:=FALSE;
				IF FBCalcPlungeGrinding.xEndWorking THEN
					iStepPrc:=400;
				ELSE
					iStepPrc:=700;
				END_IF;
			END_IF;
		(* ToolFeeder go to Start Position *)
		700:IF NOT(xInitStep) THEN
				xInitStep:=TRUE;
				TAxisToolFeeder.T_CtrleSingle.lrAcceleration:=T_Standard.T_TeachINToolFeeder.rAcceleration;
				TAxisToolFeeder.T_CtrleSingle.lrDecceleration:=T_Standard.T_TeachINToolFeeder.rDeceleration;
				TAxisToolFeeder.T_CtrleSingle.lrPosition:=T_ProcessImageData.T_ProcessPara.rStartPosToolFeedAuto;
				TAxisToolFeeder.T_CtrleSingle.lrVelocity:=T_ProcessImageData.T_ProcessPara.rSpeedStartPosToolFeedProcess;
				TAxisToolFeeder.T_CtrleSingle.iFunction:=7;	(* Move Absolut *)
				TAxisToolFeeder.T_CtrleSingle.xExecute:=TRUE;
			END_IF;
			IF NOT(TAxisToolFeeder.T_CtrleSingle.xExecute) AND TAxisToolFeeder.T_CtrleSingle.xDone THEN
				(* Only for MicroRod --> Work next cycle *)
				xStartMainPrc:=FALSE;
				xInitStep:=FALSE;
				iStepPrc:=800;
			END_IF;
		(* GrindFeeder Set Absolut to ToolDiameter minus the offset with the fast speed *)
		800:IF NOT(xInitStep) THEN
				xInitStep:=TRUE;
				TAxisGrindFeeder.T_CtrleSingle.lrAcceleration:=T_Standard.T_TeachINGrindFeeder.rAcceleration;
				TAxisGrindFeeder.T_CtrleSingle.lrDecceleration:=T_Standard.T_TeachINGrindFeeder.rDeceleration;
				TAxisGrindFeeder.T_CtrleSingle.lrPosition:=T_ProcessImageData.T_ProcessPara.rToolDiameterProcess + T_ProcessImageData.T_ProcessPara.rOffsetBeforeToolDiaGrindFeedProcess;
				TAxisGrindFeeder.T_CtrleSingle.lrVelocity:=T_ProcessImageData.T_ProcessPara.rSpeedForwardFastGrindFeed;
				TAxisGrindFeeder.T_CtrleSingle.iFunction:=7;	(* Move Absolut *)
				TAxisGrindFeeder.T_CtrleSingle.xExecute:=TRUE;
			END_IF;
			IF NOT(TAxisGrindFeeder.T_CtrleSingle.xExecute) AND TAxisGrindFeeder.T_CtrleSingle.xDone THEN
				(* Only for MicroRod --> Work next cycle *)
				xStartMainPrc:=FALSE;
				xInitStep:=FALSE;
				iStepPrc:=801;
			END_IF;
		(* GrindFeeder Set Absolut to ToolDiameter with the slow speed *)
		801:	(*IF NOT(xInitStep) THEN
				xInitStep:=TRUE;
				TAxisGrindFeeder.T_CtrleSingle.lrAcceleration:=T_Standard.T_TeachINGrindFeeder.rAcceleration;
				TAxisGrindFeeder.T_CtrleSingle.lrDecceleration:=T_Standard.T_TeachINGrindFeeder.rDeceleration;
				TAxisGrindFeeder.T_CtrleSingle.lrPosition:=T_ProcessImageData.T_ProcessPara.rToolDiameterProcess;
				TAxisGrindFeeder.T_CtrleSingle.lrVelocity:=T_ProcessImageData.T_ProcessPara.rSpeedForwardSlowGrindFeed;
				TAxisGrindFeeder.T_CtrleSingle.iFunction:=7;	(* Move Absolut *)
				TAxisGrindFeeder.T_CtrleSingle.xExecute:=TRUE;
			END_IF;
			IF NOT(TAxisGrindFeeder.T_CtrleSingle.xExecute) AND TAxisGrindFeeder.T_CtrleSingle.xDone THEN
				(* Only for MicroRod --> Work next cycle *)*)
				xStartMainPrc:=FALSE;
				xInitStep:=FALSE;
				iStepPrc:=300;
				iCountDownPlungeCycle:=iCountDownPlungeCycle + 1;
			(*END_IF;*)
		900:	xStartMainPrc:=FALSE;
			xInitStep:=FALSE;
			iStepPrc:=0;
			xSetEnd:=TRUE;
	END_CASE;
END_IF;
(******************************************************************************************************************************************)
(****************************				           Parallel Procedure Part                                          *****************************)
(******************************************************************************************************************************************)
(******************************************************************************************************************************************)
(****************************				             	Init / Reset Part                                                   *****************************)
(******************************************************************************************************************************************)
IF xSetEnd THEN
	xEnd:=TRUE;
	xInitStep:=FALSE;
	xSetEnd:=FALSE;
	xStop:=FALSE;
	xStartMainPrc:=FALSE;
	xInitMainCtr:=FALSE;
	xStartMainCtr:=FALSE;
	xStart:=FALSE;
	xHardwareError:=FALSE;
	xQuitErr:=FALSE;
	xError:=FALSE;
	iErrorNr:=0;
	xInitError:=FALSE;
	xFreeze:=FALSE;
	xAbord:=FALSE;
	xReset:=FALSE;
	xCheckToolFeedPosition:=FALSE;
	bActivePartNumber:=0;
(*	lrProcessToolFeederActualPosition:=0.0;*)
	lrProcessToolFeederSpeed:=0.0;
	rSpeedToolFeed:=0.0;
END_IF;
END_FUNCTION_BLOCK

(* POU GENERAL/FB_TOOL_CALCUL_NEW, ST *)
FUNCTION_BLOCK FB_TOOL_CALCUL_NEW
VAR_INPUT
	xMicroRodActive: BOOL;			(* choice of the machine MicroWire or MicroRod *)
	xBeckhoffDriveActive: BOOL;		(* choice of the Axis Beckhoff or EcoStep *)
	rToolFeedAcclDecl: REAL;
END_VAR
VAR_IN_OUT
	T_WorkTool:ST_WORKTOOL;		(* Tool Parameter *)
END_VAR
VAR_OUTPUT
END_VAR
VAR
	rWayAcclDecl: REAL;
	rWayConst: REAL;
	rTimeAcclDecl: REAL;
	rTimeConst: REAL;
	rTmpToolFeedAcclDecl: REAL;
	rCheckFactor: REAL;
	iTmpBaseGearDivider: INT;
	ii: INT;
	iChkNumber: INT;
END_VAR
(****************************************************************************************************************************************************)
(***********                                  This Functionblock calculate all needed parameter for work a Tool                                            ************)
(****************************************************************************************************************************************************)
(* calcul ToolRotation Speed in inc/64s *)
	IF (T_WorkTool.rToolRotationSpeed <> 0) AND (T_WorkTool.rToolRightGearRatio <> 0) THEN
		T_WorkTool.rToolRotationSpeedMotor:=((T_WorkTool.rToolRotationSpeed / 60.0) * 8000.0 * 64.0) / T_WorkTool.rToolRightGearRatio;
	ELSE
		RETURN;	(* Exit FB *)
	END_IF;
(* calcul ToolFeeder Speed in mm/s *)
	T_WorkTool.rToolFeederSpeedUnit:=T_WorkTool.rPitch * (T_WorkTool.rToolRotationSpeed / 60.0);
(* calcul ToolFeeder Speed in inc/64s Relativ *)
	T_WorkTool.rToolFeederSpeedMotorRel:=T_WorkTool.rToolFeederScaleFactor * T_WorkTool.rToolFeederSpeedUnit * 64.0;
(* calcul ToolFeeder Speed in inc/64s Relativ *)
	T_WorkTool.rToolFeederSpeedMotorAbs:=(T_WorkTool.rToolRotationSpeedMotor * T_WorkTool.rToolRightGearRatio) + T_WorkTool.rToolFeederSpeedMotorRel;
(* Set ToolFeeder GearDivider *)
	T_WorkTool.iToolFeederGearDivider:=T_WorkTool.iBaseGearDivider;
	IF xMicroRodActive THEN
	(* calcul ToolFeeder GearFactor *)
		IF (T_WorkTool.rPitch <> 0) THEN
			iTmpBaseGearDivider:=T_WorkTool.iBaseGearDivider;
			iChkNumber:=(T_WorkTool.iBaseGearDivider / 1000) - 1;	(* iBaseGearDivider is Base 15000 *)
			(* check first if the factor *)
			rCheckFactor:=INT_TO_REAL(iTmpBaseGearDivider) / (T_WorkTool.rToolRotationSpeedMotor / T_WorkTool.rToolFeederSpeedMotorRel);
			FOR ii:=1 TO iChkNumber DO
				IF (ABS(rCheckFactor) <= 32767.0) OR (iTmpBaseGearDivider = 1) THEN
					T_WorkTool.iToolFeederGearFactor:=REAL_TO_INT(INT_TO_REAL(iTmpBaseGearDivider) / (T_WorkTool.rToolRotationSpeedMotor / T_WorkTool.rToolFeederSpeedMotorRel));
					EXIT;
				ELSE
					iTmpBaseGearDivider:=iTmpBaseGearDivider - 1000;
					IF (iTmpBaseGearDivider <= 0) THEN
						iTmpBaseGearDivider:=1;
					END_IF;
					rCheckFactor:=INT_TO_REAL(iTmpBaseGearDivider) / (T_WorkTool.rToolRotationSpeedMotor / T_WorkTool.rToolFeederSpeedMotorRel);
				END_IF;
			END_FOR;
			T_WorkTool.iToolFeederGearDivider:=iTmpBaseGearDivider;
		ELSE
			T_WorkTool.iToolFeederGearFactor:=REAL_TO_INT(INT_TO_REAL(T_WorkTool.iToolFeederGearDivider) * T_WorkTool.rToolRightGearRatio);
		END_IF;
	ELSE
	(* calcul ToolFeeder GearFactor *)
		IF (T_WorkTool.rPitch <> 0) THEN
			T_WorkTool.iToolFeederGearFactor:=REAL_TO_INT(INT_TO_REAL(T_WorkTool.iBaseGearDivider) / (T_WorkTool.rToolRotationSpeedMotor / T_WorkTool.rToolFeederSpeedMotorAbs));
		ELSE
			T_WorkTool.iToolFeederGearFactor:=REAL_TO_INT(INT_TO_REAL(T_WorkTool.iToolFeederGearDivider) * T_WorkTool.rToolRightGearRatio);
		END_IF;
	END_IF;
(* calcul Time to work *)
	IF NOT(xMicroRodActive) THEN
		IF (T_WorkTool.rToolFeederSpeedUnit <> 0) THEN
			T_WorkTool.rTimeLeftWork:=(T_WorkTool.rToolLength * 10.0) / ABS(T_WorkTool.rToolFeederSpeedUnit);
		ELSE
			T_WorkTool.rTimeLeftWork:=0.0;
		END_IF;
	ELSE
		IF (T_WorkTool.rToolFeederSpeedUnit <> 0) THEN
			IF (rToolFeedAcclDecl = 0) THEN
				T_WorkTool.rTimeLeftWork:=(T_WorkTool.rToolLength * 10.0) / ABS(T_WorkTool.rToolFeederSpeedUnit);					(*calc in sec *)
			ELSE
				rTmpToolFeedAcclDecl:=rToolFeedAcclDecl * 64.0 * T_WorkTool.rToolFeederScaleFactor / 16.0;															(* calc in mm/s*s *)
				(* s_a = v^2 / 2*a *)
				rWayAcclDecl:=(T_WorkTool.rToolFeederSpeedUnit * T_WorkTool.rToolFeederSpeedUnit) / (2.0 * rTmpToolFeedAcclDecl);	(* calc in mm *)
				(* s_const = s - s_a *)
				rWayConst:=(T_WorkTool.rToolLength * 10.0) - rWayAcclDecl;														(* calc in mm *)
				IF (rWayConst <= 0) THEN	(* check if max Speed is reached *)
					(* t_a = sqrt(2*s / a) *)
					rTimeAcclDecl:=SQRT((2.0 * (T_WorkTool.rToolLength * 10.0)) / rTmpToolFeedAcclDecl);	(*calc in sec *)
					(* const velocity not reached --> t_const = 0 *)
					rTimeConst:=0.0;																	(*calc in sec *)
					(* t_total = t_a + t_const --> = t_a *)
					T_WorkTool.rTimeLeftWork:=rTimeAcclDecl + rTimeConst;								(*calc in sec *)
				ELSE
					(* t_a = sqrt(2*s_a / a) *)
					rTimeAcclDecl:=SQRT((2.0 * rWayAcclDecl) / rTmpToolFeedAcclDecl);					(*calc in sec *)
					(* t_const = s_const / v *)
					rTimeConst:=rWayConst / ABS(T_WorkTool.rToolFeederSpeedUnit);						(*calc in sec *)
					(* t_total = t_a + t_const *)
					T_WorkTool.rTimeLeftWork:=rTimeAcclDecl + rTimeConst;								(*calc in sec *)
				END_IF;
			END_IF;
		ELSE
			T_WorkTool.rTimeLeftWork:=0.0;
		END_IF;
	END_IF;
(* calcul ToolFeeder relative Position to drive *)
	T_WorkTool.rToolFeederRelPositionUnit:=T_WorkTool.rToolLength * 10.0;
	T_WorkTool.rToolFeederRelPositionMotor:=T_WorkTool.rToolFeederRelPositionUnit * T_WorkTool.rToolFeederScaleFactor;
(* calcul GrindFeeder Speed in um/s *)
	IF (T_WorkTool.rTimeLeftWork <> 0) THEN
		T_WorkTool.rGrindFeederSpeedUnit:=T_WorkTool.rGrindFeederPlunge / T_WorkTool.rTimeLeftWork;
	ELSE
		T_WorkTool.rGrindFeederSpeedUnit:=0.0;
	END_IF;
(* calcul GrindFeeder Speed in inc/s *)
	T_WorkTool.rGrindFeederSpeedMotor:=T_WorkTool.rGrindFeederSpeedUnit * T_WorkTool.rGrindFeederScaleFactor * 64.0;
END_FUNCTION_BLOCK

(* POU GENERAL/FB_CALC_GEARFACTOR, ST *)
FUNCTION_BLOCK FB_CALC_GEARFACTOR
VAR_INPUT
	rSpeed:REAL;				(* Speed in mm/s *)
	rToolRotationSpeed:REAL;		(* Speed in U/Min *)
	T_WorkTool:ST_WORKTOOL;	(* Tool Parameter *)
END_VAR
VAR_OUTPUT
END_VAR
VAR
END_VAR
(****************************************************************************************************************************************************)
(***********                                 This Functionblock calculate the gear factor for the ToolFeeder axis                                           ************)
(****************************************************************************************************************************************************)
(* Set ToolFeeder Speed in mm/s *)
	T_WorkTool.rToolFeederSpeedUnit:=rSpeed;
(* Set ToolRotation Speed in U/Min *)
	T_WorkTool.rToolRotationSpeed:=rToolRotationSpeed;
(* calcul ToolRotation Speed in inc/64s *)
	T_WorkTool.rToolRotationSpeedMotor:=((T_WorkTool.rToolRotationSpeed / 60.0) * 8000.0 * 64.0) / T_WorkTool.rToolRightGearRatio;
(* calcul ToolFeeder Speed in inc/64s Relativ *)
	T_WorkTool.rToolFeederSpeedMotorRel:=T_WorkTool.rToolFeederScaleFactor * T_WorkTool.rToolFeederSpeedUnit * 64.0;
(* calcul ToolFeeder Speed in inc/64s Relativ *)
	T_WorkTool.rToolFeederSpeedMotorAbs:=(T_WorkTool.rToolRotationSpeedMotor * T_WorkTool.rToolRightGearRatio) + T_WorkTool.rToolFeederSpeedMotorRel;
(* Set ToolFeeder GearDivider *)
	T_WorkTool.iToolFeederGearDivider:=T_WorkTool.iBaseGearDivider;
(* calcul ToolFeeder GearFactor *)
	IF (rSpeed <> 0) THEN
		T_WorkTool.iToolFeederGearFactor:=REAL_TO_INT(INT_TO_REAL(T_WorkTool.iBaseGearDivider) / (T_WorkTool.rToolRotationSpeedMotor / T_WorkTool.rToolFeederSpeedMotorAbs));
	ELSE
		T_WorkTool.iToolFeederGearFactor:=REAL_TO_INT(INT_TO_REAL(T_WorkTool.iToolFeederGearDivider) * T_WorkTool.rToolRightGearRatio);
	END_IF;
END_FUNCTION_BLOCK

(* POU PRG_STATION_LAYER3/FB_STATIONEN/FB_FUNCTION/FB_FctToolWorkingGeometryMultiCycle, ST *)
FUNCTION_BLOCK FB_FctToolWorkingGeometryMultiCycle
VAR_INPUT
	xMicroRodActive: BOOL;		(* choice of the machine MicroWire or MicroRod *)
	xBeckhoffDriveActive: BOOL;	(* choice of the axis Beckhoff or EcoStep *)
	xSafetyCircuitOn:BOOL;			(* state of the safety circuit-->TRUE=Machine current ON, FALSE=Machine current OFF *)
	T_ProcessImageData:ST_RETAIN_DATA_PROCESSIMAGE;	(* Novram data structure for the process parameter *)
	T_Standard:ST_RETAIN_DATA;							(* Novram data structure for the standard process parameter *)
END_VAR
VAR_IN_OUT
	xStart : BOOL;					(* start the function *)
	xReset : BOOL;				(* reset the function *)
	xStop : BOOL;					(* stop the active function *)
	xQuitErr : BOOL;				(* quit the error caused of the active function *)
	xAbord : BOOL;				(* abord the active function *)
	TAxisToolLeft:ST_AXIS;		(* data structure for the ToolLeft axis *)
	TAxisToolCenter:ST_AXIS;		(* data structure for the ToolCenter axis *)
	TAxisToolRight:ST_AXIS;		(* data structure for the ToolRight axis *)
	TAxisToolFeeder:ST_AXIS;		(* data structure for the ToolFeeder axis *)
	TAxisGrindFeeder:ST_AXIS;	(* data structure for the GrindFeeder axis *)
	T_WorkTool:ST_WORKTOOL;	(* Tool parameter *)
END_VAR
VAR_OUTPUT
	xEnd : BOOL;					(* state of the function if a active function is ended *)
	xError : BOOL;					(* state of the function if a active function caused an error *)
	iErrorNr : INT;					(* state of the function if a active function caused an error, in this case give the error number *)
	bActivePartNumber:BYTE;		(* gives the active number of the worked section of the geometry *)
	lrProcessToolFeederActualPosition:LREAL;	(* gives the calculated position of the ToolFeeder *)
	lrProcessToolFeederSpeed:LREAL;			(* gives the calculated speed of the ToolFeeder *)
	iCountDownPlungeCycle:INT;
END_VAR
VAR
	xHardwareError: BOOL := FALSE;
	xInitError: BOOL := FALSE;
	iStepError: INT := 0;
	xStartMainCtr: BOOL := FALSE;
	xStartMainPrc: BOOL := FALSE;
	xInitMainCtr: BOOL := FALSE;
	iStepPrc: INT := 0;
	xSetEnd: BOOL := FALSE;
	xInitStep: BOOL := FALSE;
	xFreeze: BOOL := FALSE;
	iTmpErrorNr:INT:=0;
	xTmpInit:BOOL;
	iTmp:INT;
	xTmp: BOOL;
	xReadFirstTime: BOOL;
	xTmp1: BOOL;
	rToolRotationSpeed: REAL;
	FBToolCalcul:FB_TOOL_CALCUL_NEW;

	rToolFeedLength: REAL;
	rToolDiameter: REAL;
	rGrindFeedPlunge: REAL;
	ii: INT;
	iStartSection: INT;
	iEndSection: INT;
	rSpeedGrindFeed: REAL;
	rSpeedToolFeed: REAL;
	rTimeGrindPlunge: REAL;
	FBCalcGearFactor: FB_CALC_GEARFACTOR;
	lrToolFeederActualPosition: LREAL;
	iTmpStartSection: INT;
(*22.12.2009: KFS 	{    *)
	(*
	FBCalcPlungeGrinding: FB_CALC_PLUNGE_GRINDING;
	*)
	FBCalcPlungeGrinding: FB_CALC_PLUNGE_GRINDING_MultiCycle;
	xFirstCountDownPlungeCycle:BOOL;
	xInitFB:BOOL;
	lrToolFeederStartSectionOffset: LREAL;
	xCalculationGrindingSection:BOOL;
(*22.12.2009: KFS 	}    *)
	xResetFB: BOOL;
	xGrindFeedMaster: BOOL;
	xCheckToolFeedPosition: BOOL;
	lrToolFeederPosition: LREAL;
	lrToolRightPosition: LREAL;
	lrSaveToolFeederPosition: LREAL;
	lrSaveToolRightPosition: LREAL;
	rPlungeCycleGrindFeedGeometry: REAL;
	lrGearFactor: LREAL;
	xPositionReached: BOOL;
	lrToolFeedCalcLengthPosition: REAL;
	lrCalcToolLengthInc: LREAL;
	lrCalcToolLength: LREAL;
	xReadyToolFeedStop: BOOL;
	xReadyGrindFeedStop: BOOL;
END_VAR
(****************************************************************************************************************************************************)
(***********                                This Functionblock define the function for work a geometry on the tool                                          ************)
(****************************************************************************************************************************************************)

IF NOT(xReadFirstTime) THEN
	xReadFirstTime:=TRUE;
END_IF;
(******************************************************************************************************************************************)
(****************************				           Reset Function Part                                                 *****************************)
(******************************************************************************************************************************************)
IF xReset AND NOT(xSetEnd) THEN
	xEnd:=FALSE;
	xSetEnd:=TRUE;
END_IF;
(******************************************************************************************************************************************)
(****************************				              Error Controlling Part                                            *****************************)
(******************************************************************************************************************************************)
xTmp:=	TAxisToolLeft.T_CtrleSingle.xErr OR
		(TAxisToolCenter.T_CtrleSingle.xErr AND xMicroRodActive) OR
		TAxisToolRight.T_CtrleSingle.xErr OR
		TAxisToolFeeder.T_CtrleSingle.xErr OR
		TAxisGrindFeeder.T_CtrleSingle.xErr;
xTmp1:=	NOT(TAxisToolLeft.T_CtrleSingle.xExecute) AND
		((NOT(TAxisToolCenter.T_CtrleSingle.xExecute) AND xMicroRodActive) OR NOT(xMicroRodActive)) AND
		 NOT(TAxisToolRight.T_CtrleSingle.xExecute) AND
		((NOT(TAxisToolFeeder.T_CtrleSingle.xExecute) AND NOT(xMicroRodActive)) OR xMicroRodActive) AND
		NOT(TAxisGrindFeeder.T_CtrleSingle.xExecute);
IF (xHardwareError OR (xTmp AND xStartMainPrc)) AND NOT(xSetEnd) THEN
	IF xTmp1 THEN
		IF NOT(xInitError) THEN
			iStepError:=100;
			xInitError:=TRUE;
			IF xHardwareError THEN
				iErrorNr:=iTmpErrorNr;
			ELSE
				xHardwareError:=TRUE;	(* Hardware Error *)
			END_IF;
		END_IF;
		CASE iStepError OF
			100:	iStepError:=0;
				xError:=TRUE;
		END_CASE;
		IF xQuitErr THEN
			xSetEnd:=TRUE;
		END_IF;
	END_IF;
END_IF;
(******************************************************************************************************************************************)
(****************************				              Main Controlling Part                                            *****************************)
(******************************************************************************************************************************************)
IF (xStart OR xStartMainCtr) AND NOT(xSetEnd) AND NOT(xHardwareError) THEN
	IF NOT (xInitMainCtr) THEN
		iTmpErrorNr:=0;
		iStepPrc:=100;
		xInitMainCtr:=TRUE;
		xStartMainCtr:=TRUE;
		xStart:=FALSE;
		xEnd:=FALSE;
		xAbord:=FALSE;
		xTmpInit:=FALSE;
		xCheckToolFeedPosition:=FALSE;
		bActivePartNumber:=0;
		lrCalcToolLengthInc:=lrCalcToolLength:=0.0;
		rSpeedToolFeed:=0.0;
		iCountDownPlungeCycle:=1;
	END_IF;
	IF xStop AND NOT(xTmpInit) THEN
		xTmpInit:=TRUE;
		iTmp:=100;
		RETURN;
	END_IF;
	IF xFreeze THEN
		IF xStart AND NOT(xAbord) THEN
			xFreeze:=FALSE;
			xStart:=FALSE;
		END_IF;
		IF xAbord THEN
			xAbord:=FALSE;
			xFreeze:=FALSE;
			xStart:=FALSE;
			xSetEnd:=TRUE;
		END_IF;
		RETURN;
	END_IF;
	IF NOT(xStartMainPrc) AND NOT(xSetEnd) THEN
		xStartMainPrc:=TRUE;
	END_IF;
END_IF;
(******************************************************************************************************************************************)
(****************************		               Controlling of the ToolFeeder Position                            *****************************)
(******************************************************************************************************************************************)
IF xCheckToolFeedPosition THEN
	lrToolFeederPosition:=TAxisToolFeeder.T_LiveValue.lrActualPositionNotModulo - lrSaveToolFeederPosition;
	lrToolFeederActualPosition:=(lrToolFeederPosition / TAxisToolFeeder.T_CtrleSingle.lrScaleFactor);
	lrCalcToolLength:=lrToolFeederActualPosition;
ELSE
	lrSaveToolFeederPosition:=TAxisToolFeeder.T_LiveValue.lrActualPositionNotModulo;
	lrToolFeederActualPosition:=lrToolFeederPosition:=0.0;
END_IF;
lrProcessToolFeederActualPosition:=lrCalcToolLength;
lrProcessToolFeederSpeed:=rSpeedToolFeed;
(******************************************************************************************************************************************)
(****************************				             immediate Stop Part                                              *****************************)
(******************************************************************************************************************************************)
IF xTmpInit AND NOT(xSetEnd) THEN
	IF NOT(xSafetyCircuitOn) THEN
		xTmpInit:=FALSE;
		iTmp:=100;
		xSetEnd:=TRUE;
		RETURN;
	END_IF;
	CASE iTmp OF
		100:	xReadyToolFeedStop:=xReadyGrindFeedStop:=FALSE;
			TAxisGrindFeeder.T_CtrleSingle.lrAcceleration:=T_Standard.T_TeachINToolFeeder.rAcceleration;
			TAxisGrindFeeder.T_CtrleSingle.lrDecceleration:=T_Standard.T_TeachINToolFeeder.rDeceleration;
			TAxisGrindFeeder.T_CtrleSingle.iFunction:=5;	(* Stop Movement *)
			TAxisGrindFeeder.T_CtrleSingle.xExecute:=TRUE;
			iTmp:=200;
			RETURN;
		200:	IF NOT(TAxisGrindFeeder.T_CtrleSingle.xExecute) AND TAxisGrindFeeder.T_CtrleSingle.xDone THEN
				TAxisGrindFeeder.T_CtrleSingle.lrAcceleration:=T_Standard.T_TeachINGrindFeeder.rAcceleration;
				TAxisGrindFeeder.T_CtrleSingle.lrDecceleration:=T_Standard.T_TeachINGrindFeeder.rDeceleration;
				TAxisGrindFeeder.T_CtrleSingle.lrPosition:=	T_ProcessImageData.T_ProcessPara.rToolDiameterProcess +
														T_ProcessImageData.T_ProcessPara.rSecurityPosGrindFeedProcess;
				TAxisGrindFeeder.T_CtrleSingle.lrVelocity:=T_ProcessImageData.T_ProcessPara.rSpeedBackwardGrindFeed;
				TAxisGrindFeeder.T_CtrleSingle.iFunction:=7;	(* Move Absolut *)
				TAxisGrindFeeder.T_CtrleSingle.xExecute:=TRUE;
				iTmp:=300;
			END_IF;
			RETURN;
		300:	IF NOT(TAxisGrindFeeder.T_CtrleSingle.xExecute) AND TAxisGrindFeeder.T_CtrleSingle.xDone AND NOT(xReadyGrindFeedStop) THEN
				xReadyGrindFeedStop:=TRUE;
			END_IF;
			IF (TAxisGrindFeeder.T_LiveValue.lrActualPosition >= (T_ProcessImageData.T_ProcessPara.rToolDiameterProcess + T_ProcessImageData.T_ProcessPara.rOffsetBeforeToolDiaGrindFeedProcess)) AND NOT(xReadyToolFeedStop) THEN
				xReadyToolFeedStop:=TRUE;
				xCheckToolFeedPosition:=FALSE;
				IF NOT(TAxisToolFeeder.T_CtrleSingle.xNotMoving) THEN
					TAxisToolFeeder.T_CtrleSingle.lrAcceleration:=T_Standard.T_TeachINToolFeeder.rAcceleration;
					TAxisToolFeeder.T_CtrleSingle.lrDecceleration:=T_Standard.T_TeachINToolFeeder.rDeceleration;
					TAxisToolFeeder.T_CtrleSingle.iFunction:=5;	(* Stop Movement *)
					TAxisToolFeeder.T_CtrleSingle.xExecute:=TRUE;
				END_IF;
				lrProcessToolFeederSpeed:=0.0;
			END_IF;
			IF xReadyToolFeedStop AND xReadyGrindFeedStop THEN
				iTmp:=400;
			END_IF;
			RETURN;
		400:	IF NOT(TAxisToolFeeder.T_CtrleSingle.xExecute) AND TAxisToolFeeder.T_CtrleSingle.xDone THEN
				iTmp:=500;
			END_IF;
			RETURN;
		500:	xTmpInit:=FALSE;
			iTmp:=100;
			xSetEnd:=TRUE;
			RETURN;
	END_CASE;
END_IF;
(******************************************************************************************************************************************)
(****************************				             Main Procedure Part                                             *****************************)
(******************************************************************************************************************************************)
IF xStartMainPrc AND NOT(xSetEnd) AND NOT(xHardwareError) THEN
	CASE iStepPrc OF
		(* Initial Procedure *)
		100:	rToolFeedLength:=0.0;
			rToolDiameter:=T_ProcessImageData.T_ProcessPara.rToolDiameterProcess;
			rGrindFeedPlunge:=0.0;
			rSpeedGrindFeed:=0.0;
			rSpeedToolFeed:=0.0;
			lrToolFeederStartSectionOffset:=0.0;
			iStartSection:=1;
			xInitFB:=FALSE;
			xFirstCountDownPlungeCycle:=FALSE;
			(* Check Start and End Section of the ToolGeometry *)
			FOR ii:=1 TO 6 DO
				IF T_ProcessImageData.T_GeometryPara.axActiveSection[ii] THEN
					IF (iStartSection = 0) THEN
						iStartSection:=ii;
					END_IF;
					iEndSection:=ii;
				END_IF;
			END_FOR;
			xResetFB:=TRUE;
			FBCalcPlungeGrinding(	rToolDiameter:= T_ProcessImageData.T_ProcessPara.rToolDiameterProcess,
									rToolDiameterWithOffset:=T_ProcessImageData.T_ProcessPara.rToolDiameterProcess + T_ProcessImageData.T_ProcessPara.rOffsetBeforeToolDiaGrindFeedProcess,
									xReset:= xResetFB,
									xInit:= xInitFB);
			rPlungeCycleGrindFeedGeometry:=T_ProcessImageData.T_AutoGeometryPara.rPlungeCycleGrindFeedGeometry;
			xInitFB:=TRUE;
			FBCalcPlungeGrinding(	T_Geometry:= T_ProcessImageData.T_GeometryPara,
									T_AutoGeometryPara:= T_ProcessImageData.T_AutoGeometryPara,
									rToolDiameter:= T_ProcessImageData.T_ProcessPara.rToolDiameterProcess,
									rToolDiameterWithOffset:=T_ProcessImageData.T_ProcessPara.rToolDiameterProcess + T_ProcessImageData.T_ProcessPara.rOffsetBeforeToolDiaGrindFeedProcess,
									rPlungeCycleGrindFeedGeometry:=rPlungeCycleGrindFeedGeometry,
									iStartSection:= iStartSection,
									iEndSection:= iEndSection,
									xReset:= xResetFB,
									xInit:= xInitFB);

			xStartMainPrc:=FALSE;
			xInitStep:=FALSE;
			iStepPrc:=120;
		(* Calculat the actual Start Position of ToolFeeder *)
		120:IF NOT(xInitStep) THEN
				xInitStep:=TRUE;
				FBCalcPlungeGrinding(	T_Geometry:= T_ProcessImageData.T_GeometryPara,
										T_AutoGeometryPara:= T_ProcessImageData.T_AutoGeometryPara,
										rToolDiameter:= T_ProcessImageData.T_ProcessPara.rToolDiameterProcess,
										rToolDiameterWithOffset:=T_ProcessImageData.T_ProcessPara.rToolDiameterProcess + T_ProcessImageData.T_ProcessPara.rOffsetBeforeToolDiaGrindFeedProcess,
										rPlungeCycleGrindFeedGeometry:=rPlungeCycleGrindFeedGeometry,
										iStartSection:= iStartSection,
										iEndSection:= iEndSection,
										xReset:= xResetFB,
										xInit:= xInitFB);
				xCalculationGrindingSection:=TRUE;
			END_IF;
			IF xInitStep THEN
				iTmpStartSection:=iStartSection + (FBCalcPlungeGrinding.iStepSectionWork-1);
				lrToolFeederStartSectionOffset:= 0.0;

				FOR ii:= iTmpStartSection TO  iEndSection BY 1 DO
					IF xCalculationGrindingSection THEN
						FBCalcPlungeGrinding(	T_Geometry:= T_ProcessImageData.T_GeometryPara,
												T_AutoGeometryPara:= T_ProcessImageData.T_AutoGeometryPara,
												rToolDiameter:= T_ProcessImageData.T_ProcessPara.rToolDiameterProcess,
												rToolDiameterWithOffset:=T_ProcessImageData.T_ProcessPara.rToolDiameterProcess + T_ProcessImageData.T_ProcessPara.rOffsetBeforeToolDiaGrindFeedProcess,
												rPlungeCycleGrindFeedGeometry:=rPlungeCycleGrindFeedGeometry,
												iStartSection:= iStartSection,
												iEndSection:= iEndSection,
												xReset:= xResetFB,
												xInit:= xInitFB);
						IF ( FBCalcPlungeGrinding.rActualPositionGrindFeedEnd[ii+1] <  FBCalcPlungeGrinding.rToolDiameterWithOffset ) THEN
							xCalculationGrindingSection:= FALSE;
						ELSE
							lrToolFeederStartSectionOffset:= lrToolFeederStartSectionOffset + (T_ProcessImageData.T_GeometryPara.arSectionLength[ii+1] * 10); (* Vorgabe in cm! Übergabe in mm!  --> *10 *)
						END_IF;
					END_IF;
				END_FOR;
				IF FBCalcPlungeGrinding.xEndWorking THEN
					iStepPrc:=400;
				ELSE
					IF xFirstCountDownPlungeCycle THEN
						iCountDownPlungeCycle:=iCountDownPlungeCycle + 1;
					END_IF;
					bActivePartNumber:=INT_TO_BYTE(FBCalcPlungeGrinding.iStepSectionWork);
					iStepPrc:=140;
				END_IF;
				xStartMainPrc:=FALSE;
				xInitStep:=FALSE;
			END_IF;
		(* ToolFeeder go to actual Start Position *)
		140:IF NOT(xInitStep) THEN
				xInitStep:=TRUE;
				TAxisToolFeeder.T_CtrleSingle.lrAcceleration:=T_Standard.T_TeachINToolFeeder.rAcceleration;
				TAxisToolFeeder.T_CtrleSingle.lrDecceleration:=T_Standard.T_TeachINToolFeeder.rDeceleration;
				TAxisToolFeeder.T_CtrleSingle.lrPosition:=T_ProcessImageData.T_ProcessPara.rStartPosToolFeedAuto + lrToolFeederStartSectionOffset;
				TAxisToolFeeder.T_CtrleSingle.lrVelocity:=T_ProcessImageData.T_ProcessPara.rSpeedStartPosToolFeedProcess;
				TAxisToolFeeder.T_CtrleSingle.iFunction:=7;	(* Move Absolut *)
				TAxisToolFeeder.T_CtrleSingle.xExecute:=TRUE;
			END_IF;
			IF NOT(TAxisToolFeeder.T_CtrleSingle.xExecute) AND TAxisToolFeeder.T_CtrleSingle.xDone THEN
				xStartMainPrc:=FALSE;
				xInitStep:=FALSE;
				iStepPrc:=160;
			END_IF;
		(* GrindFeeder Set Absolut to ToolDiameter minus the offset with the fast speed *)
		160:  IF NOT(xInitStep) THEN
				xInitStep:=TRUE;
				TAxisGrindFeeder.T_CtrleSingle.lrAcceleration:=T_Standard.T_TeachINGrindFeeder.rAcceleration;
				TAxisGrindFeeder.T_CtrleSingle.lrDecceleration:=T_Standard.T_TeachINGrindFeeder.rDeceleration;
				TAxisGrindFeeder.T_CtrleSingle.lrPosition:=T_ProcessImageData.T_ProcessPara.rToolDiameterProcess + T_ProcessImageData.T_ProcessPara.rOffsetBeforeToolDiaGrindFeedProcess;
				TAxisGrindFeeder.T_CtrleSingle.lrVelocity:=T_ProcessImageData.T_ProcessPara.rSpeedForwardFastGrindFeed;
				TAxisGrindFeeder.T_CtrleSingle.iFunction:=7;	(* Move Absolut *)
				TAxisGrindFeeder.T_CtrleSingle.xExecute:=TRUE;
			END_IF;
			IF NOT(TAxisGrindFeeder.T_CtrleSingle.xExecute) AND TAxisGrindFeeder.T_CtrleSingle.xDone THEN
				(* Move GrindFeed to StartPosition of actual section *)
				xStartMainPrc:=FALSE;
				xInitStep:=FALSE;
				iStepPrc:=180;
			END_IF;
		(* GrindFeeder Move to Relativ to StartDiameter of the actuel section with the slow speed *)
		180:  IF NOT(xInitStep) THEN
				xInitStep:=TRUE;
				(* StartPosition GrindFeeder wird nur solange Angefahren bis die Position direkt aus dem FBCalcPlungeGrinding berechnet wird -> iStepSection = 0 *)
				IF FBCalcPlungeGrinding.iStepSectionWork >0 THEN
					iTmpStartSection:=iStartSection + (FBCalcPlungeGrinding.iStepSectionWork - 1);
					(* Calculation of the Offset *)
					rGrindFeedPlunge:= ( FBCalcPlungeGrinding.rToolDiameterWithOffset - FBCalcPlungeGrinding.rActualPositionGrindFeedStart[iTmpStartSection] )* -1.0;
					TAxisGrindFeeder.T_CtrleSingle.lrAcceleration:=T_Standard.T_TeachINGrindFeeder.rAcceleration;
					TAxisGrindFeeder.T_CtrleSingle.lrDecceleration:=T_Standard.T_TeachINGrindFeeder.rDeceleration;
					TAxisGrindFeeder.T_CtrleSingle.lrDistance:=rGrindFeedPlunge;
					TAxisGrindFeeder.T_CtrleSingle.lrVelocity:=T_ProcessImageData.T_ProcessPara.rSpeedForwardSlowGrindFeed;
					TAxisGrindFeeder.T_CtrleSingle.iFunction:=8;	(* Move Relativ *)
					TAxisGrindFeeder.T_CtrleSingle.xExecute:=TRUE;
				END_IF;
			END_IF;
			IF NOT(TAxisGrindFeeder.T_CtrleSingle.xExecute) AND TAxisGrindFeeder.T_CtrleSingle.xDone THEN
				(* Start with AutoGeometry working *)
				xStartMainPrc:=FALSE;
				xInitStep:=FALSE;
				iStepPrc:=300;
			END_IF;
		(* Calculation of Grind plunge of all section, include Plunge procedure and Displace procedure *)
		200:	IF NOT(xInitStep) THEN
				xInitStep:=TRUE;
				FBCalcPlungeGrinding(	T_Geometry:= T_ProcessImageData.T_GeometryPara,
										T_AutoGeometryPara:= T_ProcessImageData.T_AutoGeometryPara,
										rToolDiameter:= T_ProcessImageData.T_ProcessPara.rToolDiameterProcess,
										rToolDiameterWithOffset:=T_ProcessImageData.T_ProcessPara.rToolDiameterProcess + T_ProcessImageData.T_ProcessPara.rOffsetBeforeToolDiaGrindFeedProcess,
										rPlungeCycleGrindFeedGeometry:=rPlungeCycleGrindFeedGeometry,
										iStartSection:= iStartSection,
										iEndSection:= iEndSection,
										xReset:= xResetFB,
										xInit:= xInitFB);
			END_IF;
			IF xInitStep THEN
				bActivePartNumber:=INT_TO_BYTE(FBCalcPlungeGrinding.iStepSectionWork);
				xStartMainPrc:=FALSE;
				xInitStep:=FALSE;
				IF FBCalcPlungeGrinding.xEndWorking THEN
					iStepPrc:=400;
				ELSE
					iStepPrc:=300;
				END_IF;
			END_IF;
		300:	IF NOT(xInitStep) THEN
				xInitStep:=TRUE;
				xGrindFeedMaster:=FALSE;
	(********************************                              Plunge Procedure                         *******************************)
				IF (FBCalcPlungeGrinding.iStepSectionWork = 0) THEN
(*22.12.2009: KFS 	{   *)
					rToolFeedLength:=0.0;
					rSpeedToolFeed:=0.0;
					T_WorkTool.rToolLength:=0.0;

					rSpeedGrindFeed:=T_ProcessImageData.T_AutoGeometryPara.rPlungeSpeedGrindFeedGeometry;
					rGrindFeedPlunge:=FBCalcPlungeGrinding.rGrindingRelativePosition * -1.0;

					T_WorkTool.rPitch:=T_ProcessImageData.T_GeometryPara.arSectionPitch[iStartSection] * -1.0;
					rToolRotationSpeed:=T_ProcessImageData.T_AutoGeometryPara.rSpeedToolRotationGeometry;
(*22.12.2009: KFS 	}   *)
				END_IF;
	(********************************                              Geometry Procedure                         *******************************)
				IF (FBCalcPlungeGrinding.iStepSectionWork > 0) AND (FBCalcPlungeGrinding.iStepSectionWork < 7) THEN
					(* Check first active section *)
					iTmpStartSection:=iStartSection + (FBCalcPlungeGrinding.iStepSectionWork - 1);
					T_WorkTool.rToolRotationSpeed:=T_ProcessImageData.T_AutoGeometryPara.rSpeedToolRotationGeometry;
					T_WorkTool.rPitch:=T_ProcessImageData.T_GeometryPara.arSectionPitch[iTmpStartSection] * -1.0;
					T_WorkTool.rToolLength:=T_ProcessImageData.T_GeometryPara.arSectionLength[iTmpStartSection];
					rGrindFeedPlunge:=FBCalcPlungeGrinding.rGrindingRelativePosition * -1.0;
					T_WorkTool.rGrindFeederPlunge:=rGrindFeedPlunge;
					FBToolCalcul(	xMicroRodActive:=xMicroRodActive,
									xBeckhoffDriveActive:=FALSE,
									T_WorkTool:= T_WorkTool,
									rToolFeedAcclDecl:= 0);
					rSpeedGrindFeed:=T_WorkTool.rGrindFeederSpeedUnit;
					rToolFeedLength:=T_WorkTool.rToolLength;
					rSpeedToolFeed:=T_WorkTool.rToolFeederSpeedUnit;
					rToolRotationSpeed:=T_WorkTool.rToolRotationSpeed;
				END_IF;
	(********************************                              Displace Procedure                         *******************************)
				IF (FBCalcPlungeGrinding.iStepSectionWork = 7) THEN
(*22.12.2009: KFS 	{   *)
					rToolFeedLength:=0.0;
					rSpeedToolFeed:=0.0;
					T_WorkTool.rToolLength:=0.0;

					rSpeedGrindFeed:=T_ProcessImageData.T_AutoGeometryPara.rDisplaceSpeedGrindFeedGeometry;
					rGrindFeedPlunge:=FBCalcPlungeGrinding.rGrindingRelativePosition * -1.0;

					T_WorkTool.rPitch:=T_ProcessImageData.T_GeometryPara.arSectionPitch[iEndSection] * -1.0;
					rToolRotationSpeed:=T_ProcessImageData.T_AutoGeometryPara.rSpeedToolRotationGeometry;
(*22.12.2009: KFS 	}   *)
				END_IF;
	(********************************                              Drive Procedure                             *******************************)
				IF (*TAxisToolFeeder.T_CtrleSingle.xNotMoving AND*) (rToolFeedLength <> 0) THEN
					TAxisToolFeeder.T_CtrleSingle.lrAcceleration:=T_Standard.T_TeachINToolFeeder.rAcceleration;
					TAxisToolFeeder.T_CtrleSingle.lrDecceleration:=T_Standard.T_TeachINToolFeeder.rDeceleration;
					IF (FBCalcPlungeGrinding.iStepSectionWork > 0) AND (FBCalcPlungeGrinding.iStepSectionWork < 7) THEN
						TAxisToolFeeder.T_CtrleSingle.lrVelocity:=rSpeedToolFeed * -1.0;
					ELSE
						TAxisToolFeeder.T_CtrleSingle.lrVelocity:=rSpeedToolFeed;
					END_IF;
					TAxisToolFeeder.T_CtrleSingle.iFunction:=6;	(* Move continue velocity *)
					TAxisToolFeeder.T_CtrleSingle.xExecute:=TRUE;
				END_IF;
				IF NOT(TAxisToolFeeder.T_CtrleSingle.xNotMoving) AND (rToolFeedLength = 0) THEN
					TAxisToolFeeder.T_CtrleSingle.lrAcceleration:=T_Standard.T_TeachINToolFeeder.rAcceleration;
					TAxisToolFeeder.T_CtrleSingle.lrDecceleration:=T_Standard.T_TeachINToolFeeder.rDeceleration;
					TAxisToolFeeder.T_CtrleSingle.iFunction:=5;	(* Stop Movement *)
					TAxisToolFeeder.T_CtrleSingle.xExecute:=TRUE;
				END_IF;
				(* Start GrindFeeder *)
				IF (rGrindFeedPlunge <> 0) THEN
					xGrindFeedMaster:=TRUE;
					IF (rToolFeedLength <> 0) THEN
						xCheckToolFeedPosition:=TRUE;	(* Start Measure Relative Position of the ToolFeeder *)
					END_IF;
					IF (FBCalcPlungeGrinding.iStepSectionWork > 0) THEN
						TAxisGrindFeeder.T_CtrleSingle.xBlockAcclDeclParameter:=TRUE;	(* do not send again the accl and decl parameter-->better performance *)
					END_IF;
					TAxisGrindFeeder.T_CtrleSingle.lrAcceleration:=T_Standard.T_TeachINGrindFeeder.rAcceleration;
					TAxisGrindFeeder.T_CtrleSingle.lrDecceleration:=T_Standard.T_TeachINGrindFeeder.rDeceleration;
					TAxisGrindFeeder.T_CtrleSingle.lrDistance:=rGrindFeedPlunge;
					TAxisGrindFeeder.T_CtrleSingle.lrVelocity:=rSpeedGrindFeed;
					TAxisGrindFeeder.T_CtrleSingle.iFunction:=8;	(* Move Relative *)
					TAxisGrindFeeder.T_CtrleSingle.xExecute:=TRUE;
				ELSE
					xGrindFeedMaster:=FALSE;
					xCheckToolFeedPosition:=TRUE;	(* Start Measure Relative Position of the ToolFeeder *)
				END_IF;
			END_IF;
	(********************************                              Wait end active section                             *******************************)
			IF xGrindFeedMaster THEN
			(* This is active by plunge procedure or displace procedure or by work a cone section *)
				IF NOT(TAxisGrindFeeder.T_CtrleSingle.xExecute) AND TAxisGrindFeeder.T_CtrleSingle.xDone THEN
					xCheckToolFeedPosition:=FALSE;
					xStartMainPrc:=FALSE;
					xInitStep:=FALSE;
					IF (FBCalcPlungeGrinding.iStepSectionWork <> 7) THEN
						iStepPrc:=200;
					ELSE
						iStepPrc:=400;
					END_IF;
				END_IF;
			END_IF;
			IF NOT(xGrindFeedMaster) THEN
			(* This is only active if it is work a cylinder section *)
				IF (lrToolFeederActualPosition > (rToolFeedLength * 10.0)) THEN
					xCheckToolFeedPosition:=FALSE;
					xStartMainPrc:=FALSE;
					xInitStep:=FALSE;
					IF (FBCalcPlungeGrinding.iStepSectionWork <> 7) THEN
						iStepPrc:=200;
					ELSE
						iStepPrc:=400;
					END_IF;
				END_IF;
			END_IF;
		(* Check if ToolFeeder Moves and stop it if it moves *)
		400:	IF NOT(xInitStep) THEN
				xInitStep:=TRUE;
				IF NOT(TAxisToolFeeder.T_CtrleSingle.xNotMoving) THEN
					TAxisToolFeeder.T_CtrleSingle.lrAcceleration:=T_Standard.T_TeachINToolFeeder.rAcceleration;
					TAxisToolFeeder.T_CtrleSingle.lrDecceleration:=T_Standard.T_TeachINToolFeeder.rDeceleration;
					TAxisToolFeeder.T_CtrleSingle.iFunction:=5;	(* Stop Movement *)
					TAxisToolFeeder.T_CtrleSingle.xExecute:=TRUE;
				END_IF;
			END_IF;
			IF NOT(TAxisToolFeeder.T_CtrleSingle.xExecute) AND TAxisToolFeeder.T_CtrleSingle.xDone THEN
				rSpeedToolFeed:=0.0;
				xStartMainPrc:=FALSE;
				xInitStep:=FALSE;
				iStepPrc:=500;
			END_IF;
		(* GrindFeeder go to Security Position *)
		500:	IF NOT(xInitStep) THEN
				xInitStep:=TRUE;
				TAxisGrindFeeder.T_CtrleSingle.lrAcceleration:=T_Standard.T_TeachINGrindFeeder.rAcceleration;
				TAxisGrindFeeder.T_CtrleSingle.lrDecceleration:=T_Standard.T_TeachINGrindFeeder.rDeceleration;
				TAxisGrindFeeder.T_CtrleSingle.lrPosition:=	T_ProcessImageData.T_ProcessPara.rToolDiameterProcess +
														T_ProcessImageData.T_ProcessPara.rSecurityPosGrindFeedProcess;
				TAxisGrindFeeder.T_CtrleSingle.lrVelocity:=T_ProcessImageData.T_ProcessPara.rSpeedBackwardGrindFeed;
				TAxisGrindFeeder.T_CtrleSingle.iFunction:=7;	(* Move Absolut *)
				TAxisGrindFeeder.T_CtrleSingle.xExecute:=TRUE;
			END_IF;
			IF NOT(TAxisGrindFeeder.T_CtrleSingle.xExecute) AND TAxisGrindFeeder.T_CtrleSingle.xDone THEN
				IF FBCalcPlungeGrinding.xEndWorking THEN
					(* Procedure is finished *)
					xStartMainPrc:=FALSE;
					xInitStep:=FALSE;
					iStepPrc:=600;
				ELSE
(*					iCountDownPlungeCycle:=iCountDownPlungeCycle + 1;*)
					xFirstCountDownPlungeCycle:=TRUE;
					xStartMainPrc:=FALSE;
					xInitStep:=FALSE;
					iStepPrc:=120;
				END_IF;
			END_IF;
		600:	xStartMainPrc:=FALSE;
			xInitStep:=FALSE;
			iStepPrc:=0;
			xSetEnd:=TRUE;
	END_CASE;
END_IF;
(******************************************************************************************************************************************)
(****************************				           Parallel Procedure Part                                          *****************************)
(******************************************************************************************************************************************)
(******************************************************************************************************************************************)
(****************************				             	Init / Reset Part                                                   *****************************)
(******************************************************************************************************************************************)
IF xSetEnd THEN
	xEnd:=TRUE;
	xInitStep:=FALSE;
	xSetEnd:=FALSE;
	xStop:=FALSE;
	xStartMainPrc:=FALSE;
	xInitMainCtr:=FALSE;
	xStartMainCtr:=FALSE;
	xStart:=FALSE;
	xHardwareError:=FALSE;
	xQuitErr:=FALSE;
	xError:=FALSE;
	iErrorNr:=0;
	xInitError:=FALSE;
	xFreeze:=FALSE;
	xAbord:=FALSE;
	xReset:=FALSE;
	xCheckToolFeedPosition:=FALSE;
	bActivePartNumber:=0;
(*	lrProcessToolFeederActualPosition:=0.0;*)
	lrProcessToolFeederSpeed:=0.0;
	rSpeedToolFeed:=0.0;
END_IF;
END_FUNCTION_BLOCK

(* POU PRG_STATION_LAYER3/FB_STATIONEN/FB_FUNCTION/FB_FctToolWorkingGroove, ST *)
FUNCTION_BLOCK FB_FctToolWorkingGroove
VAR_INPUT
	xMicroRodActive: BOOL;		(* choice of the machine MicroWire or MicroRod *)
	xBeckhoffDriveActive: BOOL;	(* choice of the axis Beckhoff or EcoStep *)
	xSafetyCircuitOn:BOOL;			(* state of the safety circuit-->TRUE=Machine current ON, FALSE=Machine current OFF *)
	xDoNotMoveGrindPosition:BOOL;							(* TRUE=override the position of the GrindAxis with the ToolDiameter, FALSE=no overriding *)
	T_ProcessImageData:ST_RETAIN_DATA_PROCESSIMAGE;	(* Novram data structure for the process parameter *)
	T_Standard:ST_RETAIN_DATA;							(* Novram data structure for the standard process parameter *)
END_VAR
VAR_IN_OUT
	xStart : BOOL;					(* start the function *)
	xReset : BOOL;				(* reset the function *)
	xStop : BOOL;					(* stop the active function *)
	xQuitErr : BOOL;				(* quit the error caused of the active function *)
	xAbord : BOOL;				(* abord the active function *)
	TAxisToolLeft:ST_AXIS;		(* data structure for the ToolLeft axis *)
	TAxisToolCenter:ST_AXIS;		(* data structure for the ToolCenter axis *)
	TAxisToolRight:ST_AXIS;		(* data structure for the ToolRight axis *)
	TAxisToolFeeder:ST_AXIS;		(* data structure for the ToolFeeder axis *)
	TAxisGrindFeeder:ST_AXIS;	(* data structure for the GrindFeeder axis *)
	T_WorkTool:ST_WORKTOOL;	(* Tool parameter *)
	(* KFS 03.09.2010* { *)
	rStartPosAutoGrooveToolRotation:REAL;
	(* KFS 03.09.2010* { *)
END_VAR
VAR_OUTPUT
	xEnd : BOOL;					(* state of the function if a active function is ended *)
	xError : BOOL;					(* state of the function if a active function caused an error *)
	iErrorNr : INT;					(* state of the function if a active function caused an error, in this case give the error number *)
	bActivePartNumber:BYTE;		(* gives the active number of the worked section of the geometry *)
	lrProcessToolFeederActualPosition:LREAL;	(* gives the calculated position of the ToolFeeder *)
	lrProcessToolFeederSpeed:LREAL;			(* gives the calculated speed of the ToolFeeder *)
END_VAR
VAR
	xHardwareError: BOOL := FALSE;
	xInitError: BOOL := FALSE;
	iStepError: INT := 0;
	xStartMainCtr: BOOL := FALSE;
	xStartMainPrc: BOOL := FALSE;
	xInitMainCtr: BOOL := FALSE;
	iStepPrc: INT := 0;
	xSetEnd: BOOL := FALSE;
	xInitStep: BOOL := FALSE;
	xFreeze: BOOL := FALSE;
	iTmpErrorNr:INT:=0;
	xTmpInit:BOOL;
	iTmp:INT;
	xTmp: BOOL;
	xReadFirstTime: BOOL;
	xTmp1: BOOL;
	rToolRotationSpeed: REAL;
	FBToolCalcul:FB_TOOL_CALCUL_NEW;

	rToolFeedLength: REAL;
	rToolDiameter: REAL;
	rGrindFeedPlunge: REAL;
	ii: INT;
	iStartSection: INT;
	iEndSection: INT;
	rSpeedGrindFeed: REAL;
	rSpeedToolFeed: REAL;
	rTimeGrindPlunge: REAL;
	FBCalcGearFactor: FB_CALC_GEARFACTOR;
	lrToolFeederActualPosition: LREAL;
	iTmpStartSection: INT;
	FBCalcPlungeGrinding: FB_CALC_PLUNGE_GRINDING;
	xResetFB: BOOL;
	xGrindFeedMaster: BOOL;
	xCheckToolFeedPosition: BOOL;
	lrToolFeederPosition: LREAL;
	lrToolRightPosition: LREAL;
	lrSaveToolFeederPosition: LREAL;
	lrSaveToolRightPosition: LREAL;
	rPlungeCycleGrindFeedGeometry: REAL;
	lrToolFeedCalcLengthPosition: REAL;
	lrCalcToolLengthInc: LREAL;
	lrCalcToolLength: LREAL;
	xReadyToolFeedStop: BOOL;
	xReadyGrindFeedStop: BOOL;
	xCheckWithoutToolRotation: BOOL;
	lrSavePos: LREAL;
END_VAR
(****************************************************************************************************************************************************)
(***********                                    This Functionblock define the function for work a groove on the tool                                          ************)
(****************************************************************************************************************************************************)

